FUNCTION_BLOCK "sq_carousel_st1"   // FB39, GRAPH
VERSION : 0.1
// stored: AcknowledgeErrorsRequired true, AutoNumber true, GraphVersion 6.0, InitialValuesAcquisition false, IsIECCheckEnabled false, LanguageInNetworks LAD, LockOperatingMode false, PermanentILProcessingInMANMode false, SetENOAutomatically false, SkipSteps false, UDAEnableTagReadback false, WithAlarmHandling true
   // inherited from GRAPH_BASE
   VAR
      OFF_SQ_BASE : Bool;
   END_VAR
   VAR_INPUT
      OFF_SQ { ExternalAccessible := 'False'; ExternalVisible := 'False'; ExternalWritable := 'False'} : Bool := false;   // Turn sequence off
      INIT_SQ { ExternalAccessible := 'False'; ExternalVisible := 'False'; ExternalWritable := 'False'} : Bool := false;   // Set sequence to initial state
      ACK_EF { ExternalAccessible := 'False'; ExternalVisible := 'False'; ExternalWritable := 'False'} : Bool := false;   // Acknowledge all errors and faults
      S_PREV { ExternalAccessible := 'False'; ExternalVisible := 'False'; ExternalWritable := 'False'} : Bool := false;   // Output previous step in parameter S_NO
      S_NEXT { ExternalAccessible := 'False'; ExternalVisible := 'False'; ExternalWritable := 'False'} : Bool := false;   // Indicate next step in parameter S_NO
      SW_AUTO { ExternalAccessible := 'False'; ExternalVisible := 'False'; ExternalWritable := 'False'} : Bool := false;   // Automatic mode
      SW_TAP { ExternalAccessible := 'False'; ExternalVisible := 'False'; ExternalWritable := 'False'} : Bool := false;   // Semiautomatic/switch with transition
      SW_TOP { ExternalAccessible := 'False'; ExternalVisible := 'False'; ExternalWritable := 'False'} : Bool := false;   // Semiautomatic/ignore transition
      SW_MAN { ExternalAccessible := 'False'; ExternalVisible := 'False'; ExternalWritable := 'False'} : Bool := false;   // Manual mode
      S_SEL { ExternalAccessible := 'False'; ExternalVisible := 'False'; ExternalWritable := 'False'} : Int := 0;   // Select step to be output to S_NO
      S_ON { ExternalAccessible := 'False'; ExternalVisible := 'False'; ExternalWritable := 'False'} : Bool := false;   // Activate step indicated in S_NO
      S_OFF { ExternalAccessible := 'False'; ExternalVisible := 'False'; ExternalWritable := 'False'} : Bool := false;   // Deactivate step indicated S_NO
      T_PUSH { ExternalAccessible := 'False'; ExternalVisible := 'False'; ExternalWritable := 'False'} : Bool := false;   // Enable transition to switch in semi automatic mode
   END_VAR
   VAR_OUTPUT
      S_NO { ExternalAccessible := 'False'; ExternalVisible := 'False'; ExternalWritable := 'False'} : Int := 0;   // Step number
      S_MORE { ExternalAccessible := 'False'; ExternalVisible := 'False'; ExternalWritable := 'False'} : Bool := false;   // More steps are available and can be shown in S_NO
      S_ACTIVE { ExternalAccessible := 'False'; ExternalVisible := 'False'; ExternalWritable := 'False'} : Bool := false;   // Step indicated in S_NO is active
      ERR_FLT { ExternalAccessible := 'False'; ExternalVisible := 'False'; ExternalWritable := 'False'} : Bool := false;   // Interlock or supervision group error
      AUTO_ON { ExternalAccessible := 'False'; ExternalVisible := 'False'; ExternalWritable := 'False'} : Bool := false;   // Automatic mode is active
      TAP_ON { ExternalAccessible := 'False'; ExternalVisible := 'False'; ExternalWritable := 'False'} : Bool := false;   // Semiautomatic mode/step with transition enabled
      TOP_ON { ExternalAccessible := 'False'; ExternalVisible := 'False'; ExternalWritable := 'False'} : Bool := false;   // Semiautomatic mode/ignore transition enabled
      MAN_ON { ExternalAccessible := 'False'; ExternalVisible := 'False'; ExternalWritable := 'False'} : Bool := false;   // Manual mode is active
   END_VAR
   VAR
      dummy : Bool;
      start : Bool;
      base : Bool;
      startEmpty : Bool;
   END_VAR
   VAR_TEMP   // added for the SCL form of the ladder/FBD networks
      _w1 : Bool;
      _w2 : Bool;
   END_VAR
BEGIN
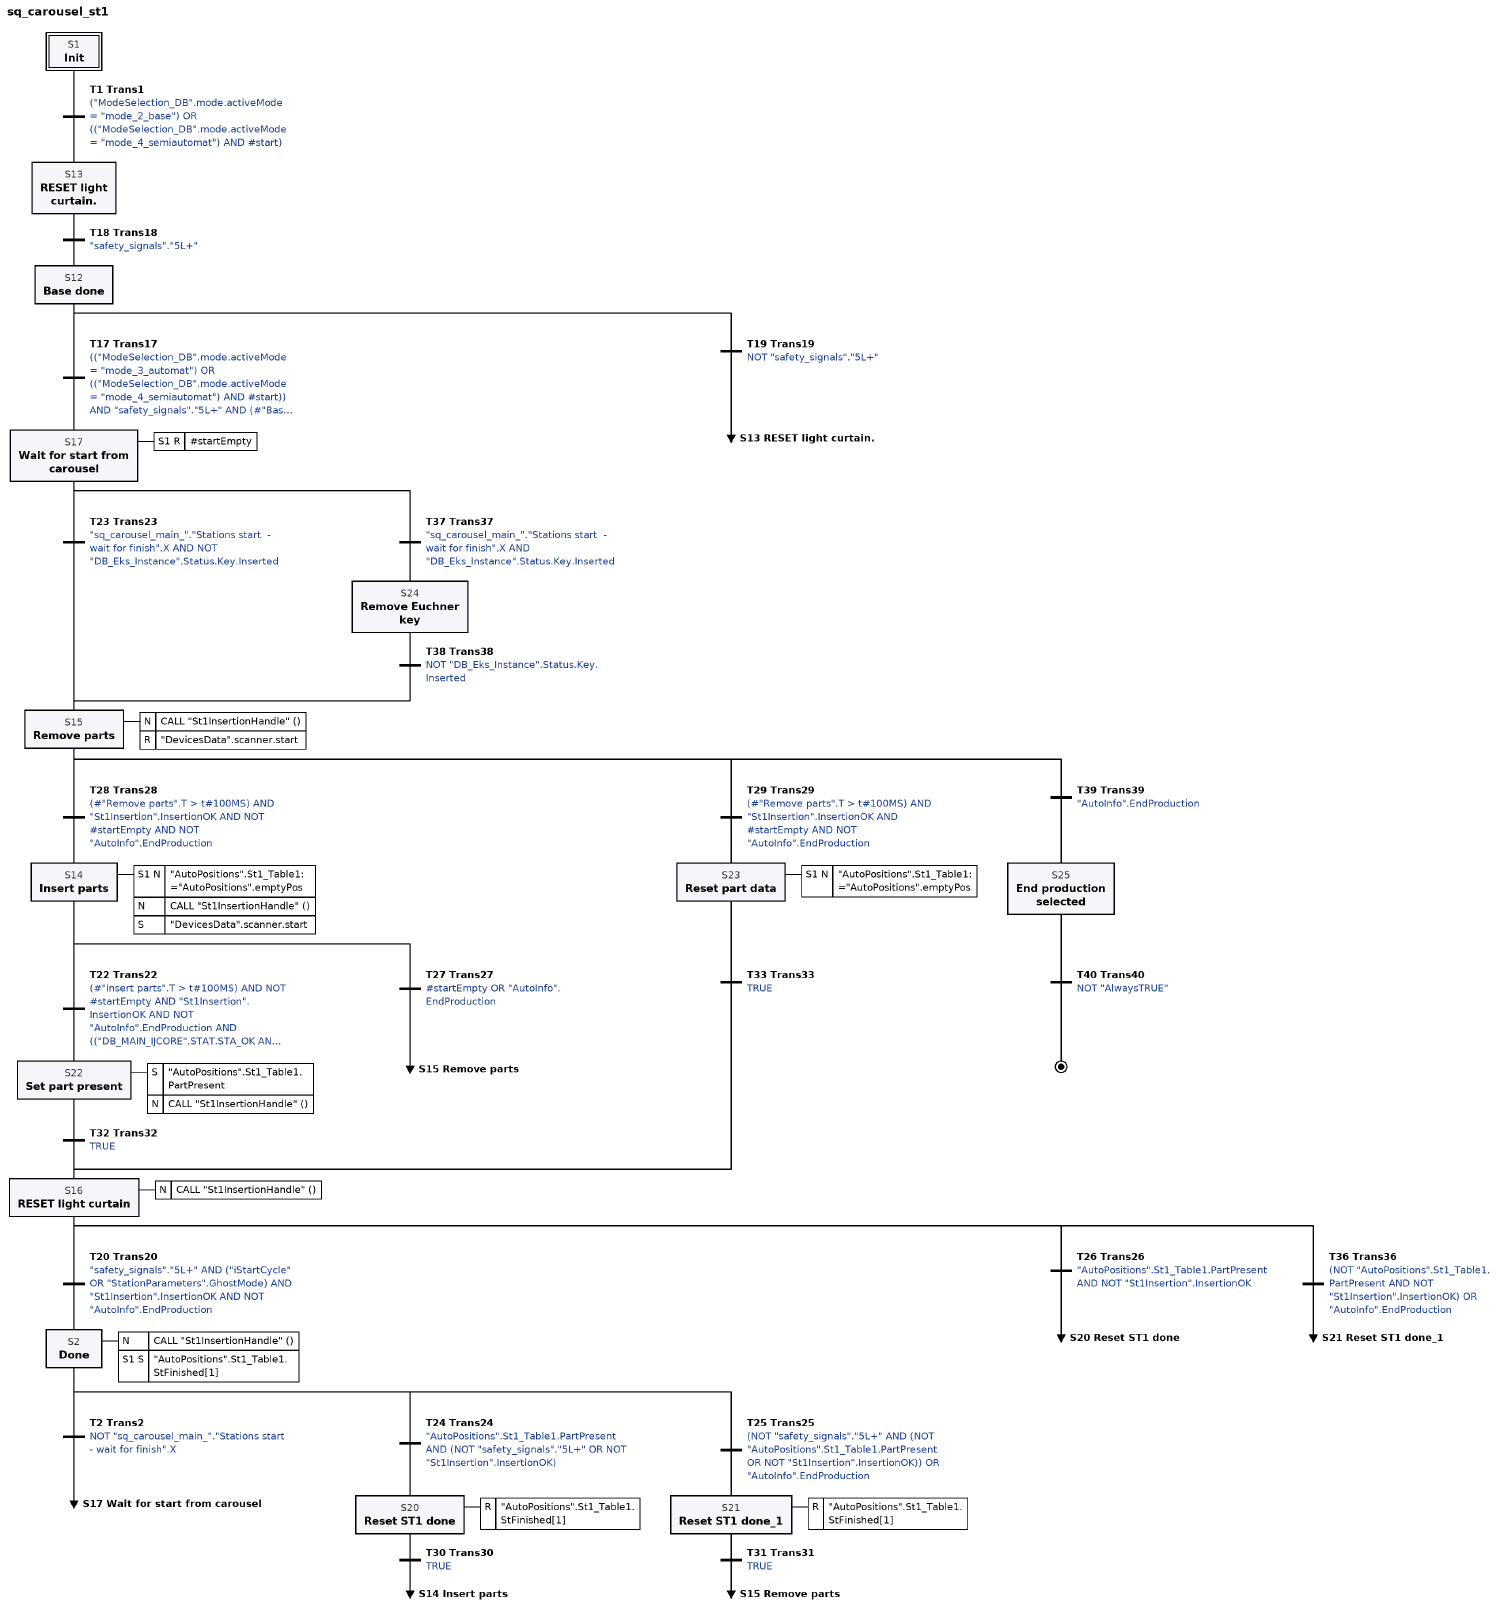
   // permanent pre-instructions
   NETWORK 1
      #base := TRUE;
   NETWORK 2
      "St1Insertion".ExpectedSensors := "St1Insertion".EmptyBits;
      #_w1 := ("ModeSelection_DB".mode.activeMode = "mode_3_automat") OR ("ModeSelection_DB".mode.activeMode = "mode_4_semiautomat");
      IF #_w1 THEN "St1Insertion".UsedSensors := "St1Insertion".FullBits; END_IF;
      IF NOT #_w1 THEN "St1Insertion".UsedSensors := "St1Insertion".EmptyBits; END_IF;
      #_w2 := ("AutoPositions".St1_Table1.PartPresent OR #"Insert parts".X) AND NOT #startEmpty AND NOT "StationParameters".GhostMode AND NOT #"Remove parts".X;
      IF #_w2 THEN
          MOVE_BLK(IN := "DB_ProductionProgramActual".Program.St1Insertion[1],
                   COUNT := 20,
                   OUT => "St1Insertion".ExpectedSensors[1]);
          MOVE_BLK(IN := "DB_ProductionProgramActual".Program.St1InsertionUsed[1],
                   COUNT := 20,
                   OUT => "St1Insertion".UsedSensors[1]);
      END_IF;
      "St1InsertionHandle"();

   // sequencer 1
   INITIAL_STEP Init:   // S1, max time T#10S, warning time T#7S
   END_STEP
   TRANSITION Trans1 FROM Init TO "RESET light curtain."   // T1
      := ("ModeSelection_DB".mode.activeMode = "mode_2_base") OR (("ModeSelection_DB".mode.activeMode = "mode_4_semiautomat") AND #start);
   END_TRANSITION
   STEP Done:   // S2, max time T#10S, warning time T#7S
              N    CALL "St1InsertionHandle" ()
          S1  S    "AutoPositions".St1_Table1.StFinished[1]
   END_STEP
   TRANSITION Trans2 FROM Done TO "Wait for start from carousel"   // T2, jump
      := NOT "sq_carousel_main_"."Stations start  - wait for finish".X;
   END_TRANSITION
   TRANSITION Trans24 FROM Done TO "Reset ST1 done"   // T24
      := "AutoPositions".St1_Table1.PartPresent AND (NOT "safety_signals"."5L+" OR NOT "St1Insertion".InsertionOK);
   END_TRANSITION
   TRANSITION Trans25 FROM Done TO "Reset ST1 done_1"   // T25
      := (NOT "safety_signals"."5L+" AND (NOT "AutoPositions".St1_Table1.PartPresent OR NOT "St1Insertion".InsertionOK)) OR "AutoInfo".EndProduction;
   END_TRANSITION
   STEP "Base done":   // S12, max time T#10S, warning time T#7S
   END_STEP
   TRANSITION Trans17 FROM "Base done" TO "Wait for start from carousel"   // T17
      := (("ModeSelection_DB".mode.activeMode = "mode_3_automat") OR (("ModeSelection_DB".mode.activeMode = "mode_4_semiautomat") AND #start)) AND "safety_signals"."5L+" AND (#"Base done".T > t#2000MS);
   END_TRANSITION
   TRANSITION Trans19 FROM "Base done" TO "RESET light curtain."   // T19, jump
      := NOT "safety_signals"."5L+";
   END_TRANSITION
   STEP "RESET light curtain.":   // S13, max time T#10S, warning time T#7S
   END_STEP
   TRANSITION Trans18 FROM "RESET light curtain." TO "Base done"   // T18
      := "safety_signals"."5L+";
   END_TRANSITION
   STEP "Insert parts":   // S14, max time T#10S, warning time T#7S
          S1  N    "AutoPositions".St1_Table1:="AutoPositions".emptyPos
              N    CALL "St1InsertionHandle" ()
              S    "DevicesData".scanner.start
   END_STEP
   TRANSITION Trans22 FROM "Insert parts" TO "Set part present"   // T22
      := (#"Insert parts".T > t#100MS) AND NOT #startEmpty AND "St1Insertion".InsertionOK AND NOT "AutoInfo".EndProduction AND (("DB_MAIN_IJCORE".STAT.STA_OK AND "DB_MAIN_IJCORE".STAT.TRC_OK) OR NOT "DB_MAIN_IJCORE".Enable);
   END_TRANSITION
   TRANSITION Trans27 FROM "Insert parts" TO "Remove parts"   // T27, jump
      := #startEmpty OR "AutoInfo".EndProduction;
   END_TRANSITION
   STEP "Remove parts":   // S15, max time T#10S, warning time T#7S
              N    CALL "St1InsertionHandle" ()
              R    "DevicesData".scanner.start
   END_STEP
   TRANSITION Trans28 FROM "Remove parts" TO "Insert parts"   // T28
      := (#"Remove parts".T > t#100MS) AND "St1Insertion".InsertionOK AND NOT #startEmpty AND NOT "AutoInfo".EndProduction;
   END_TRANSITION
   TRANSITION Trans29 FROM "Remove parts" TO "Reset part data"   // T29
      := (#"Remove parts".T > t#100MS) AND "St1Insertion".InsertionOK AND #startEmpty AND NOT "AutoInfo".EndProduction;
   END_TRANSITION
   TRANSITION Trans39 FROM "Remove parts" TO "End production selected"   // T39
      := "AutoInfo".EndProduction;
   END_TRANSITION
   STEP "RESET light curtain":   // S16, max time T#10S, warning time T#7S
              N    CALL "St1InsertionHandle" ()
   END_STEP
   TRANSITION Trans20 FROM "RESET light curtain" TO Done   // T20
      := "safety_signals"."5L+" AND ("iStartCycle" OR "StationParameters".GhostMode) AND "St1Insertion".InsertionOK AND NOT "AutoInfo".EndProduction;
   END_TRANSITION
   TRANSITION Trans26 FROM "RESET light curtain" TO "Reset ST1 done"   // T26, jump
      := "AutoPositions".St1_Table1.PartPresent AND NOT "St1Insertion".InsertionOK;
   END_TRANSITION
   TRANSITION Trans36 FROM "RESET light curtain" TO "Reset ST1 done_1"   // T36, jump
      := (NOT "AutoPositions".St1_Table1.PartPresent AND NOT "St1Insertion".InsertionOK) OR "AutoInfo".EndProduction;
   END_TRANSITION
   STEP "Wait for start from carousel":   // S17, max time T#10S, warning time T#7S
          S1  R    #startEmpty
   END_STEP
   TRANSITION Trans23 FROM "Wait for start from carousel" TO "Remove parts"   // T23
      := "sq_carousel_main_"."Stations start  - wait for finish".X AND NOT "DB_Eks_Instance".Status.Key.Inserted;
   END_TRANSITION
   TRANSITION Trans37 FROM "Wait for start from carousel" TO "Remove Euchner key"   // T37
      := "sq_carousel_main_"."Stations start  - wait for finish".X AND "DB_Eks_Instance".Status.Key.Inserted;
   END_TRANSITION
   STEP "Reset ST1 done":   // S20, max time T#10S, warning time T#7S
              R    "AutoPositions".St1_Table1.StFinished[1]
   END_STEP
   TRANSITION Trans30 FROM "Reset ST1 done" TO "Insert parts"   // T30, jump
      := TRUE;
   END_TRANSITION
   STEP "Reset ST1 done_1":   // S21, max time T#10S, warning time T#7S
              R    "AutoPositions".St1_Table1.StFinished[1]
   END_STEP
   TRANSITION Trans31 FROM "Reset ST1 done_1" TO "Remove parts"   // T31, jump
      := TRUE;
   END_TRANSITION
   STEP "Set part present":   // S22, max time T#10S, warning time T#7S
              S    "AutoPositions".St1_Table1.PartPresent
              N    CALL "St1InsertionHandle" ()
   END_STEP
   TRANSITION Trans32 FROM "Set part present" TO "RESET light curtain"   // T32
      := TRUE;
   END_TRANSITION
   STEP "Reset part data":   // S23, max time T#10S, warning time T#7S
          S1  N    "AutoPositions".St1_Table1:="AutoPositions".emptyPos
   END_STEP
   TRANSITION Trans33 FROM "Reset part data" TO "RESET light curtain"   // T33
      := TRUE;
   END_TRANSITION
   STEP "Remove Euchner key":   // S24, max time T#10S, warning time T#7S
   END_STEP
   TRANSITION Trans38 FROM "Remove Euchner key" TO "Remove parts"   // T38
      := NOT "DB_Eks_Instance".Status.Key.Inserted;
   END_TRANSITION
   STEP "End production selected":   // S25, max time T#10S, warning time T#7S
   END_STEP
   TRANSITION Trans40 FROM "End production selected" TO END   // T40
      := NOT "AlwaysTRUE";
   END_TRANSITION
END_FUNCTION_BLOCK

FUNCTION "St1InsertionHandle" : Void
{ S7_Optimized_Access := 'TRUE' }
VERSION : 0.1
   VAR_TEMP 
      i : Int;
      res : Bool;
      empty : Bool;
      lastNOKIndex : Int;
   END_VAR


BEGIN
	
	#i := 1;
	"St1Insertion".SensorsState[#i] := "DevicesData".Camera[1].Result = 1;
	#i := #i + 1;
	"St1Insertion".SensorsState[#i] := "DevicesData".Camera[2].Result = 1;
	#i := #i + 1;
	"St1Insertion".SensorsState[#i] := "DevicesData".Camera[3].Result = 1;
	#i := #i + 1;
	"St1Insertion".SensorsState[#i] := "DevicesData".Camera[4].Result = 1;
	#i := #i + 1;
	"St1Insertion".SensorsState[#i] := "DB_INST_READINGS".Reading[1].OK = 1;
	#i := #i + 1;
	"St1Insertion".SensorsState[#i] := "DB_INST_READINGS".Reading[2].OK = 1;
	#i := #i + 1;
	"St1Insertion".SensorsState[#i] := "DB_INST_READINGS".Reading[3].OK = 1;
	#i := #i + 1;
	"St1Insertion".SensorsState[#i] := "DB_INST_READINGS".Reading[4].OK = 1;
	#i := #i + 1;
	"St1Insertion".SensorsState[#i] := "DB_INST_READINGS".Reading[5].OK = 1;
	#i := #i + 1;
	"St1Insertion".SensorsState[#i] := "DB_INST_READINGS".Reading[6].OK = 1;
	#i := #i + 1;
	"St1Insertion".SensorsState[#i] := "DB_INST_READINGS".Reading[7].OK = 1;
	#i := #i + 1;
	"St1Insertion".SensorsState[#i] := "DB_INST_READINGS".Reading[8].OK = 1;
	#i := #i + 1;
	"St1Insertion".SensorsState[#i] := FALSE;
	#i := #i + 1;
	"St1Insertion".SensorsState[#i] := FALSE;
	#i := #i + 1;
	"St1Insertion".SensorsState[#i] := FALSE;
	#i := #i + 1;
	"St1Insertion".SensorsState[#i] := FALSE;
	#i := #i + 1;
	"St1Insertion".SensorsState[#i] := FALSE;
	#i := #i + 1;
	"St1Insertion".SensorsState[#i] := "Sensor_LH_PP" = 1;
	#i := #i + 1;
	"St1Insertion".SensorsState[#i] := "Sensor_RH_PP" = 1;
	
	#lastNOKIndex := 1;
	
	#res := TRUE;
	#empty := true;
	FOR #i := 1 TO 20 DO
	    
	    //Check if all sensors are zero
	    IF "St1Insertion".SensorsState[#i] THEN
	        #empty := false;
	    END_IF;
	    //Check if sensor is correct
	    IF ("St1Insertion".SensorsState[#i] <> "St1Insertion".ExpectedSensors[#i]) AND
	            "St1Insertion".UsedSensors[#i] THEN
	            #res := false;
	            "St1Insertion".SensorsNOK[#i] := true;
	            "St1Insertion".NOKList[#lastNOKIndex] := #i;
	            #lastNOKIndex := #lastNOKIndex + 1;
	        ELSE
	            "St1Insertion".SensorsNOK[#i] := false;
	    END_IF;
	END_FOR;
	    
	//Reset rest of nok list
	FOR #i := #lastNOKIndex TO 20 DO
	        "St1Insertion".NOKList[#i] := 0;
	END_FOR;
	
	"St1Insertion".InsertionOK := #res;
	"St1Insertion".InsertionNOK := NOT #empty AND NOT #res;
	"St1Insertion".InsertionEmpty := #empty;
	
	
	
END_FUNCTION

FUNCTION_BLOCK "sq_carousel_st2"   // FB43, GRAPH
VERSION : 0.1
// stored: AcknowledgeErrorsRequired true, AutoNumber true, GraphVersion 6.0, InitialValuesAcquisition false, IsIECCheckEnabled false, LanguageInNetworks LAD, LockOperatingMode false, PermanentILProcessingInMANMode false, SetENOAutomatically false, SkipSteps false, UDAEnableTagReadback false, WithAlarmHandling true
   // inherited from GRAPH_BASE
   VAR
      OFF_SQ_BASE : Bool;
   END_VAR
   VAR_INPUT
      OFF_SQ { ExternalAccessible := 'False'; ExternalVisible := 'False'; ExternalWritable := 'False'} : Bool := false;   // Turn sequence off
      INIT_SQ { ExternalAccessible := 'False'; ExternalVisible := 'False'; ExternalWritable := 'False'} : Bool := false;   // Set sequence to initial state
      ACK_EF { ExternalAccessible := 'False'; ExternalVisible := 'False'; ExternalWritable := 'False'} : Bool := false;   // Acknowledge all errors and faults
      S_PREV { ExternalAccessible := 'False'; ExternalVisible := 'False'; ExternalWritable := 'False'} : Bool := false;   // Output previous step in parameter S_NO
      S_NEXT { ExternalAccessible := 'False'; ExternalVisible := 'False'; ExternalWritable := 'False'} : Bool := false;   // Indicate next step in parameter S_NO
      SW_AUTO { ExternalAccessible := 'False'; ExternalVisible := 'False'; ExternalWritable := 'False'} : Bool := false;   // Automatic mode
      SW_TAP { ExternalAccessible := 'False'; ExternalVisible := 'False'; ExternalWritable := 'False'} : Bool := false;   // Semiautomatic/switch with transition
      SW_TOP { ExternalAccessible := 'False'; ExternalVisible := 'False'; ExternalWritable := 'False'} : Bool := false;   // Semiautomatic/ignore transition
      SW_MAN { ExternalAccessible := 'False'; ExternalVisible := 'False'; ExternalWritable := 'False'} : Bool := false;   // Manual mode
      S_SEL { ExternalAccessible := 'False'; ExternalVisible := 'False'; ExternalWritable := 'False'} : Int := 0;   // Select step to be output to S_NO
      S_ON { ExternalAccessible := 'False'; ExternalVisible := 'False'; ExternalWritable := 'False'} : Bool := false;   // Activate step indicated in S_NO
      S_OFF { ExternalAccessible := 'False'; ExternalVisible := 'False'; ExternalWritable := 'False'} : Bool := false;   // Deactivate step indicated S_NO
      T_PUSH { ExternalAccessible := 'False'; ExternalVisible := 'False'; ExternalWritable := 'False'} : Bool := false;   // Enable transition to switch in semi automatic mode
   END_VAR
   VAR_OUTPUT
      S_NO { ExternalAccessible := 'False'; ExternalVisible := 'False'; ExternalWritable := 'False'} : Int := 0;   // Step number
      S_MORE { ExternalAccessible := 'False'; ExternalVisible := 'False'; ExternalWritable := 'False'} : Bool := false;   // More steps are available and can be shown in S_NO
      S_ACTIVE { ExternalAccessible := 'False'; ExternalVisible := 'False'; ExternalWritable := 'False'} : Bool := false;   // Step indicated in S_NO is active
      ERR_FLT { ExternalAccessible := 'False'; ExternalVisible := 'False'; ExternalWritable := 'False'} : Bool := false;   // Interlock or supervision group error
      AUTO_ON { ExternalAccessible := 'False'; ExternalVisible := 'False'; ExternalWritable := 'False'} : Bool := false;   // Automatic mode is active
      TAP_ON { ExternalAccessible := 'False'; ExternalVisible := 'False'; ExternalWritable := 'False'} : Bool := false;   // Semiautomatic mode/step with transition enabled
      TOP_ON { ExternalAccessible := 'False'; ExternalVisible := 'False'; ExternalWritable := 'False'} : Bool := false;   // Semiautomatic mode/ignore transition enabled
      MAN_ON { ExternalAccessible := 'False'; ExternalVisible := 'False'; ExternalWritable := 'False'} : Bool := false;   // Manual mode is active
   END_VAR
   VAR
      dummy : Bool;
      start : Bool;
      base : Bool;
   END_VAR
BEGIN
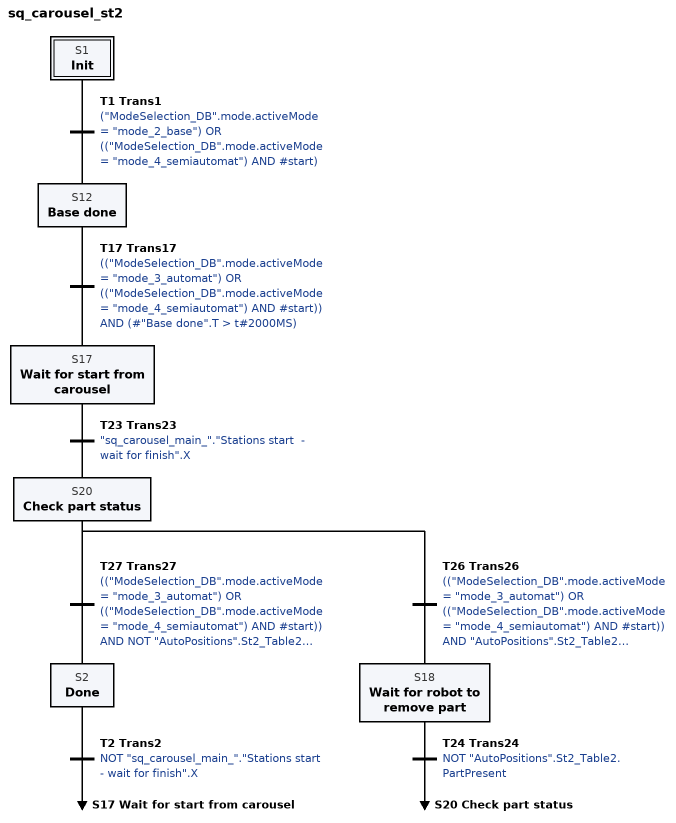
   // permanent pre-instructions
   NETWORK 1
   TITLE = base position
      #base := TRUE;

   // sequencer 1
   INITIAL_STEP Init:   // S1, max time T#10S, warning time T#7S
   END_STEP
   TRANSITION Trans1 FROM Init TO "Base done"   // T1
      := ("ModeSelection_DB".mode.activeMode = "mode_2_base") OR (("ModeSelection_DB".mode.activeMode = "mode_4_semiautomat") AND #start);
   END_TRANSITION
   STEP Done:   // S2, max time T#10S, warning time T#7S
   END_STEP
   TRANSITION Trans2 FROM Done TO "Wait for start from carousel"   // T2, jump
      := NOT "sq_carousel_main_"."Stations start  - wait for finish".X;
   END_TRANSITION
   STEP "Base done":   // S12, max time T#10S, warning time T#7S
   END_STEP
   TRANSITION Trans17 FROM "Base done" TO "Wait for start from carousel"   // T17
      := (("ModeSelection_DB".mode.activeMode = "mode_3_automat") OR (("ModeSelection_DB".mode.activeMode = "mode_4_semiautomat") AND #start)) AND (#"Base done".T > t#2000MS);
   END_TRANSITION
   STEP "Wait for start from carousel":   // S17, max time T#10S, warning time T#7S
   END_STEP
   TRANSITION Trans23 FROM "Wait for start from carousel" TO "Check part status"   // T23
      := "sq_carousel_main_"."Stations start  - wait for finish".X;
   END_TRANSITION
   STEP "Check part status":   // S20, max time T#10S, warning time T#7S
   END_STEP
   TRANSITION Trans27 FROM "Check part status" TO Done   // T27
      := (("ModeSelection_DB".mode.activeMode = "mode_3_automat") OR (("ModeSelection_DB".mode.activeMode = "mode_4_semiautomat") AND #start)) AND NOT "AutoPositions".St2_Table2.PartPresent AND "iR1OutOfSt2";
   END_TRANSITION
   TRANSITION Trans26 FROM "Check part status" TO "Wait for robot to remove part"   // T26
      := (("ModeSelection_DB".mode.activeMode = "mode_3_automat") OR (("ModeSelection_DB".mode.activeMode = "mode_4_semiautomat") AND #start)) AND "AutoPositions".St2_Table2.PartPresent;
   END_TRANSITION
   STEP "Wait for robot to remove part":   // S18, max time T#10S, warning time T#7S
   END_STEP
   TRANSITION Trans24 FROM "Wait for robot to remove part" TO "Check part status"   // T24, jump
      := NOT "AutoPositions".St2_Table2.PartPresent;
   END_TRANSITION
END_FUNCTION_BLOCK

FUNCTION_BLOCK "sq_jig"   // FB41, GRAPH
VERSION : 0.1
// stored: AcknowledgeErrorsRequired true, AutoNumber true, GraphVersion 6.0, InitialValuesAcquisition false, IsIECCheckEnabled false, LanguageInNetworks LAD, LockOperatingMode false, PermanentILProcessingInMANMode false, SetENOAutomatically false, SkipSteps false, UDAEnableTagReadback false, WithAlarmHandling true
   // inherited from GRAPH_BASE
   VAR
      OFF_SQ_BASE : Bool;
   END_VAR
   VAR_INPUT
      OFF_SQ { ExternalAccessible := 'False'; ExternalVisible := 'False'; ExternalWritable := 'False'} : Bool := false;   // Turn sequence off
      INIT_SQ { ExternalAccessible := 'False'; ExternalVisible := 'False'; ExternalWritable := 'False'} : Bool := false;   // Set sequence to initial state
      ACK_EF { ExternalAccessible := 'False'; ExternalVisible := 'False'; ExternalWritable := 'False'} : Bool := false;   // Acknowledge all errors and faults
      S_PREV { ExternalAccessible := 'False'; ExternalVisible := 'False'; ExternalWritable := 'False'} : Bool := false;   // Output previous step in parameter S_NO
      S_NEXT { ExternalAccessible := 'False'; ExternalVisible := 'False'; ExternalWritable := 'False'} : Bool := false;   // Indicate next step in parameter S_NO
      SW_AUTO { ExternalAccessible := 'False'; ExternalVisible := 'False'; ExternalWritable := 'False'} : Bool := false;   // Automatic mode
      SW_TAP { ExternalAccessible := 'False'; ExternalVisible := 'False'; ExternalWritable := 'False'} : Bool := false;   // Semiautomatic/switch with transition
      SW_TOP { ExternalAccessible := 'False'; ExternalVisible := 'False'; ExternalWritable := 'False'} : Bool := false;   // Semiautomatic/ignore transition
      SW_MAN { ExternalAccessible := 'False'; ExternalVisible := 'False'; ExternalWritable := 'False'} : Bool := false;   // Manual mode
      S_SEL { ExternalAccessible := 'False'; ExternalVisible := 'False'; ExternalWritable := 'False'} : Int := 0;   // Select step to be output to S_NO
      S_ON { ExternalAccessible := 'False'; ExternalVisible := 'False'; ExternalWritable := 'False'} : Bool := false;   // Activate step indicated in S_NO
      S_OFF { ExternalAccessible := 'False'; ExternalVisible := 'False'; ExternalWritable := 'False'} : Bool := false;   // Deactivate step indicated S_NO
      T_PUSH { ExternalAccessible := 'False'; ExternalVisible := 'False'; ExternalWritable := 'False'} : Bool := false;   // Enable transition to switch in semi automatic mode
   END_VAR
   VAR_OUTPUT
      S_NO { ExternalAccessible := 'False'; ExternalVisible := 'False'; ExternalWritable := 'False'} : Int := 0;   // Step number
      S_MORE { ExternalAccessible := 'False'; ExternalVisible := 'False'; ExternalWritable := 'False'} : Bool := false;   // More steps are available and can be shown in S_NO
      S_ACTIVE { ExternalAccessible := 'False'; ExternalVisible := 'False'; ExternalWritable := 'False'} : Bool := false;   // Step indicated in S_NO is active
      ERR_FLT { ExternalAccessible := 'False'; ExternalVisible := 'False'; ExternalWritable := 'False'} : Bool := false;   // Interlock or supervision group error
      AUTO_ON { ExternalAccessible := 'False'; ExternalVisible := 'False'; ExternalWritable := 'False'} : Bool := false;   // Automatic mode is active
      TAP_ON { ExternalAccessible := 'False'; ExternalVisible := 'False'; ExternalWritable := 'False'} : Bool := false;   // Semiautomatic mode/step with transition enabled
      TOP_ON { ExternalAccessible := 'False'; ExternalVisible := 'False'; ExternalWritable := 'False'} : Bool := false;   // Semiautomatic mode/ignore transition enabled
      MAN_ON { ExternalAccessible := 'False'; ExternalVisible := 'False'; ExternalWritable := 'False'} : Bool := false;   // Manual mode is active
   END_VAR
   VAR
      dummy : Bool;
      start : Bool;
      base : Bool;
   END_VAR
   VAR_TEMP   // added for the SCL form of the ladder/FBD networks
      _w1 : Bool;
   END_VAR
BEGIN
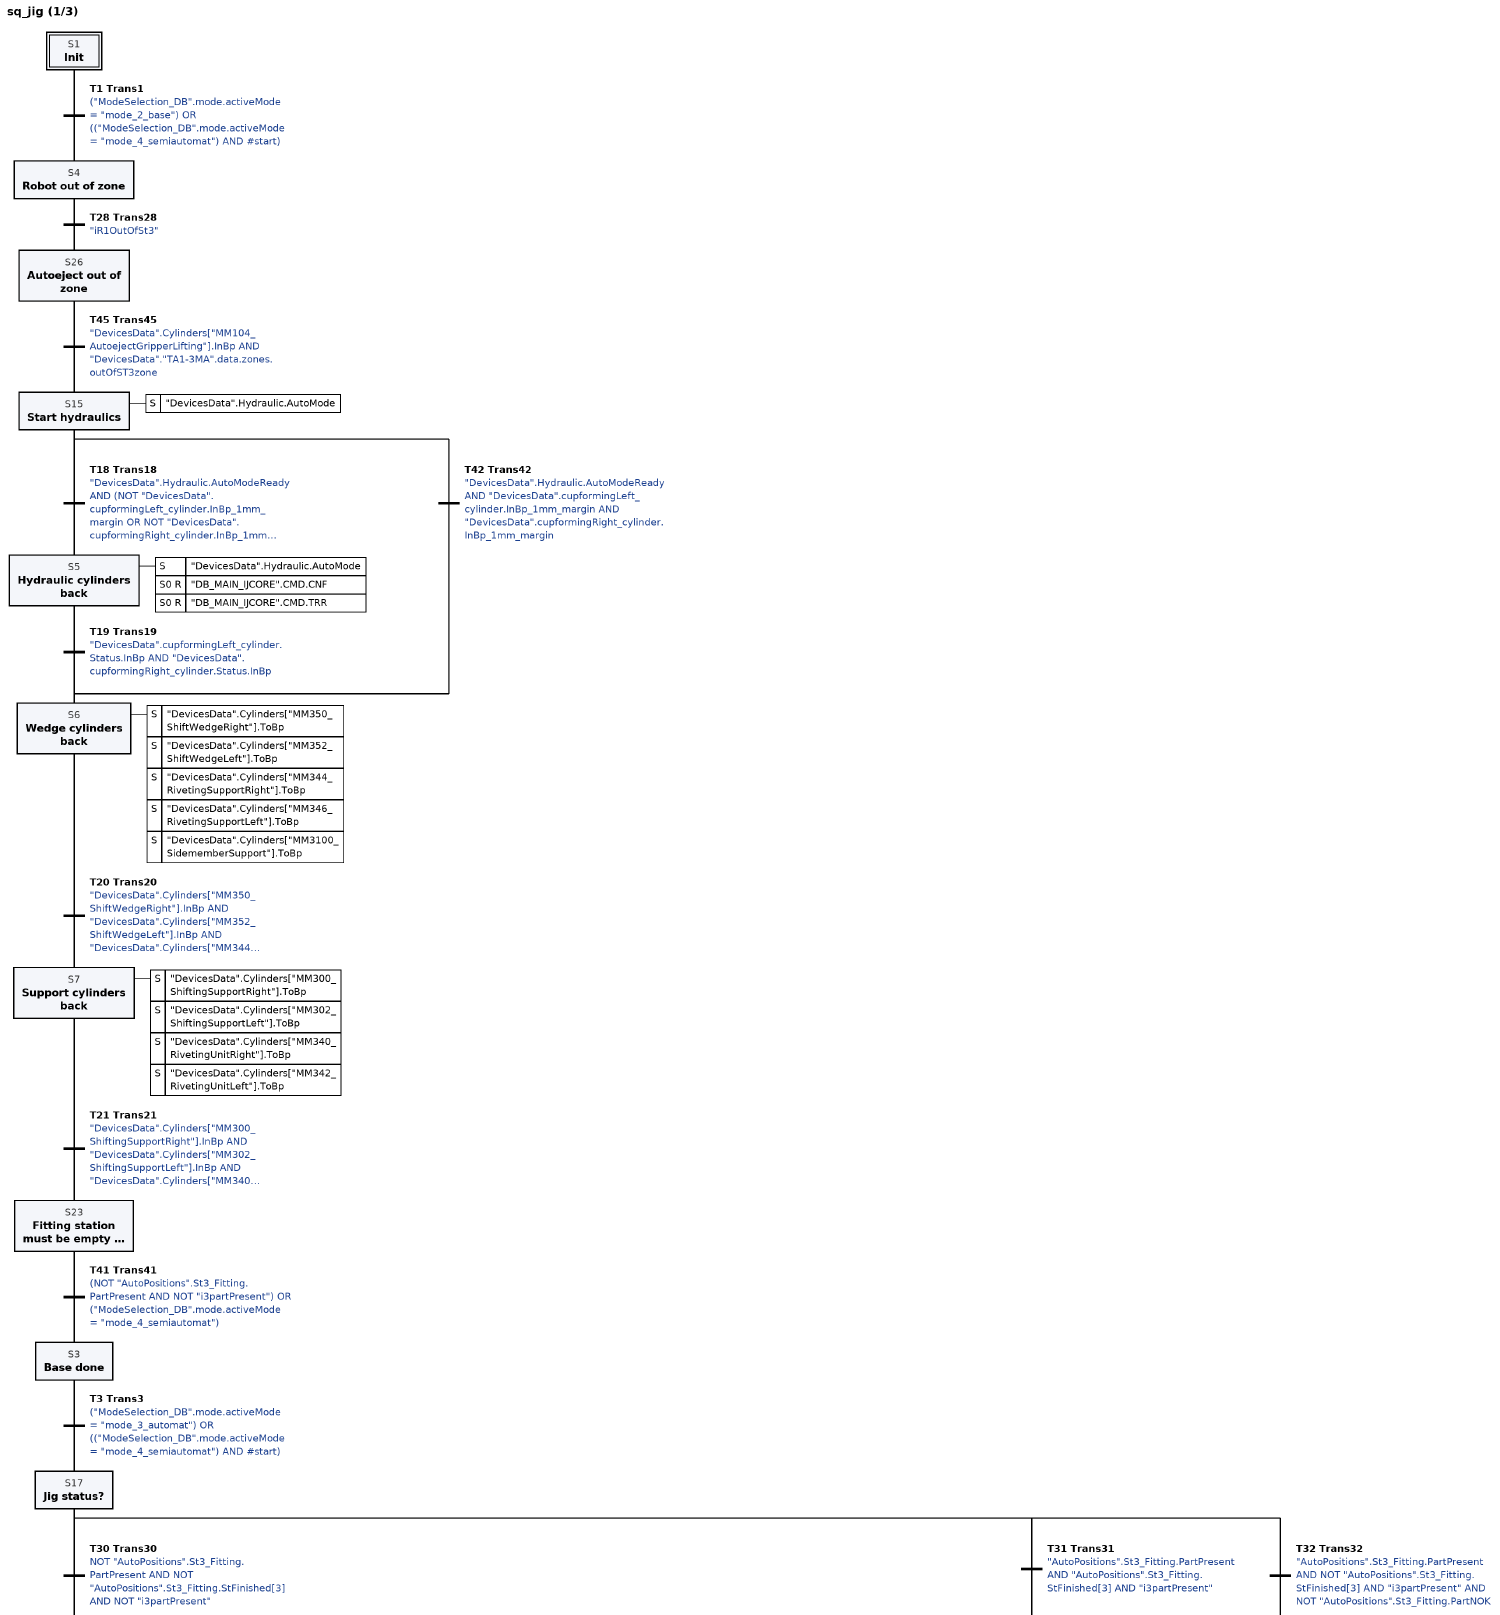
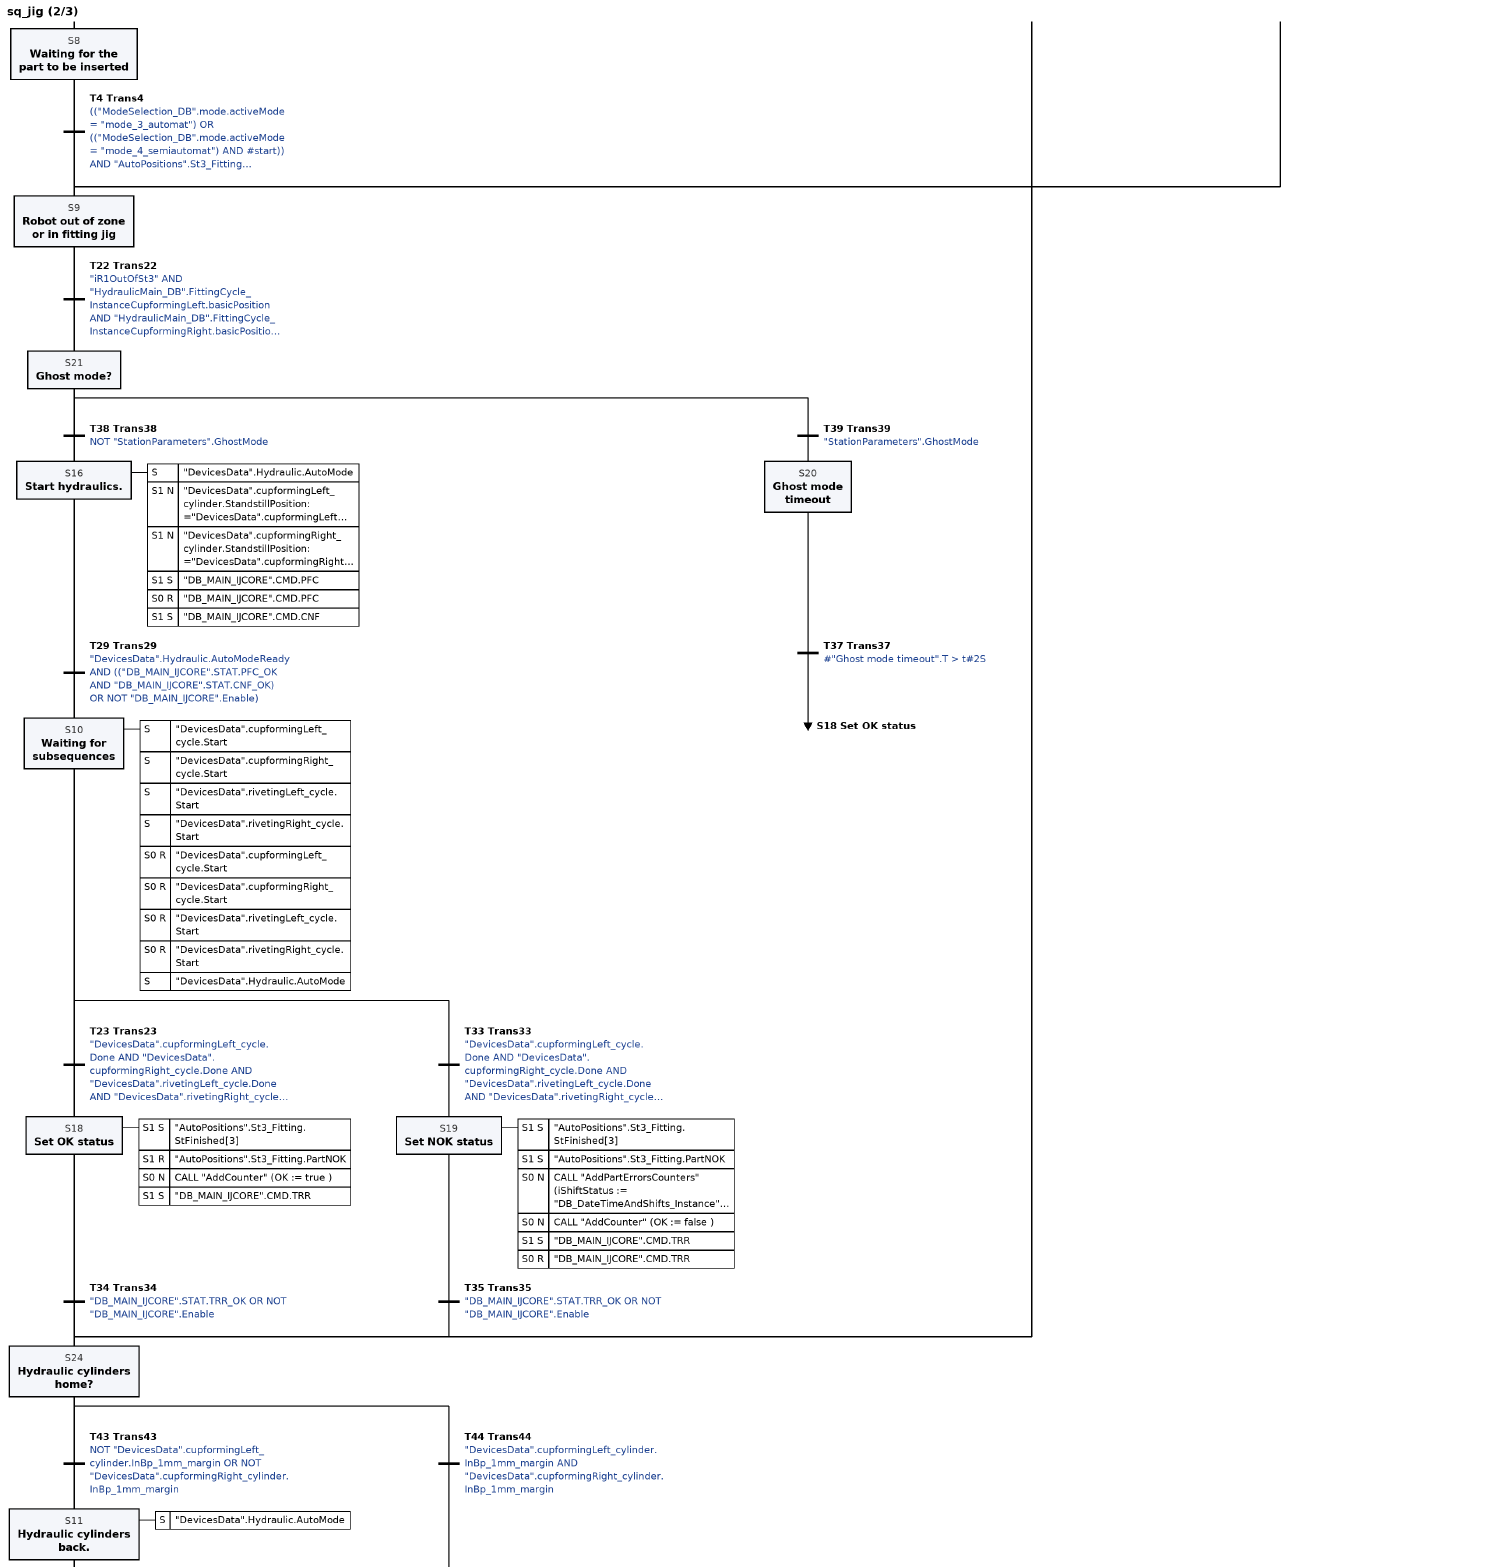
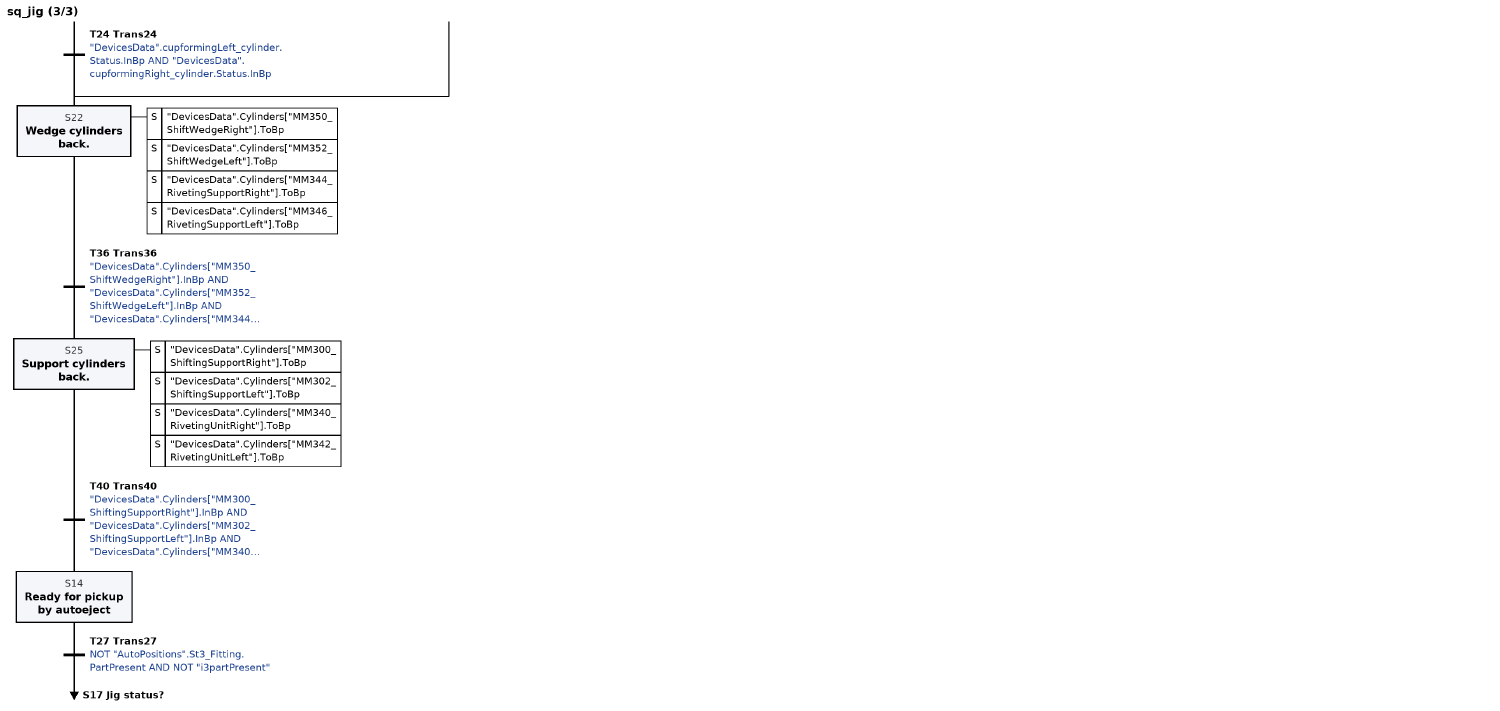
   // permanent pre-instructions
   NETWORK 1
   TITLE = base position
      #base := "HydraulicMain_DB".FittingCycle_InstanceCupformingLeft.basicPosition AND "HydraulicMain_DB".FittingCycle_InstanceCupformingRight.basicPosition AND "DB_Devices_Instance".RivetingCycleLeft_Instance.basicPosition AND "DB_Devices_Instance".RivetingCycleRight_Instance.basicPosition AND "DevicesData".Digiforce1.Ready AND "DevicesData".Digiforce1.programOK AND "DevicesData".Digiforce2.Ready AND "DevicesData".Digiforce2.programOK AND NOT "Devices_Diagnostic_DB".PNmissing;

   // sequencer 1
   INITIAL_STEP Init:   // S1, max time T#10S, warning time T#7S
   END_STEP
   TRANSITION Trans1 FROM Init TO "Robot out of zone"   // T1
      := ("ModeSelection_DB".mode.activeMode = "mode_2_base") OR (("ModeSelection_DB".mode.activeMode = "mode_4_semiautomat") AND #start);
   END_TRANSITION
   STEP "Start hydraulics":   // S15, max time T#10S, warning time T#7S
      supervision V := #"Start hydraulics".T > #"Start hydraulics".T_MAX;
              S    "DevicesData".Hydraulic.AutoMode
   END_STEP
   TRANSITION Trans18 FROM "Start hydraulics" TO "Hydraulic cylinders back"   // T18
      := "DevicesData".Hydraulic.AutoModeReady AND (NOT "DevicesData".cupformingLeft_cylinder.InBp_1mm_margin OR NOT "DevicesData".cupformingRight_cylinder.InBp_1mm_margin);
   END_TRANSITION
   TRANSITION Trans42 FROM "Start hydraulics" TO "Wedge cylinders back"   // T42
      := "DevicesData".Hydraulic.AutoModeReady AND "DevicesData".cupformingLeft_cylinder.InBp_1mm_margin AND "DevicesData".cupformingRight_cylinder.InBp_1mm_margin;
   END_TRANSITION
   STEP "Waiting for the part to be inserted":   // S8, max time T#10S, warning time T#7S
   END_STEP
   TRANSITION Trans4 FROM "Waiting for the part to be inserted" TO "Robot out of zone or in fitting jig"   // T4
      := (("ModeSelection_DB".mode.activeMode = "mode_3_automat") OR (("ModeSelection_DB".mode.activeMode = "mode_4_semiautomat") AND #start)) AND "AutoPositions".St3_Fitting.PartPresent AND NOT "AutoPositions".St3_Fitting.StFinished[3] AND ("i3partPresent" OR "StationParameters".GhostMode);
   END_TRANSITION
   STEP "Robot out of zone":   // S4, max time T#10S, warning time T#7S
      supervision V := #"Robot out of zone".T > #"Robot out of zone".T_MAX;
   END_STEP
   TRANSITION Trans28 FROM "Robot out of zone" TO "Autoeject out of zone"   // T28
      := "iR1OutOfSt3";
   END_TRANSITION
   STEP "Hydraulic cylinders back":   // S5, max time T#10S, warning time T#7S
      supervision V := #"Hydraulic cylinders back".T > #"Hydraulic cylinders back".T_MAX;
              S    "DevicesData".Hydraulic.AutoMode
          S0  R    "DB_MAIN_IJCORE".CMD.CNF
          S0  R    "DB_MAIN_IJCORE".CMD.TRR
   END_STEP
   TRANSITION Trans19 FROM "Hydraulic cylinders back" TO "Wedge cylinders back"   // T19
      := "DevicesData".cupformingLeft_cylinder.Status.InBp AND "DevicesData".cupformingRight_cylinder.Status.InBp;
   END_TRANSITION
   STEP "Wedge cylinders back":   // S6, max time T#10S, warning time T#7S
      supervision V := #"Wedge cylinders back".T > #"Wedge cylinders back".T_MAX;
              S    "DevicesData".Cylinders["MM350_ShiftWedgeRight"].ToBp
              S    "DevicesData".Cylinders["MM352_ShiftWedgeLeft"].ToBp
              S    "DevicesData".Cylinders["MM344_RivetingSupportRight"].ToBp
              S    "DevicesData".Cylinders["MM346_RivetingSupportLeft"].ToBp
              S    "DevicesData".Cylinders["MM3100_SidememberSupport"].ToBp
   END_STEP
   TRANSITION Trans20 FROM "Wedge cylinders back" TO "Support cylinders back"   // T20
      := "DevicesData".Cylinders["MM350_ShiftWedgeRight"].InBp AND "DevicesData".Cylinders["MM352_ShiftWedgeLeft"].InBp AND "DevicesData".Cylinders["MM344_RivetingSupportRight"].InBp AND "DevicesData".Cylinders["MM346_RivetingSupportLeft"].InBp AND "DevicesData".Cylinders["MM3100_SidememberSupport"].InBp;
   END_TRANSITION
   STEP "Support cylinders back":   // S7, max time T#10S, warning time T#7S
      supervision V := #"Support cylinders back".T > #"Support cylinders back".T_MAX;
              S    "DevicesData".Cylinders["MM300_ShiftingSupportRight"].ToBp
              S    "DevicesData".Cylinders["MM302_ShiftingSupportLeft"].ToBp
              S    "DevicesData".Cylinders["MM340_RivetingUnitRight"].ToBp
              S    "DevicesData".Cylinders["MM342_RivetingUnitLeft"].ToBp
   END_STEP
   TRANSITION Trans21 FROM "Support cylinders back" TO "Fitting station must be empty - remove part and delete status"   // T21
      := "DevicesData".Cylinders["MM300_ShiftingSupportRight"].InBp AND "DevicesData".Cylinders["MM302_ShiftingSupportLeft"].InBp AND "DevicesData".Cylinders["MM340_RivetingUnitRight"].InBp AND "DevicesData".Cylinders["MM342_RivetingUnitLeft"].InBp;
   END_TRANSITION
   STEP "Base done":   // S3, max time T#10S, warning time T#7S
   END_STEP
   TRANSITION Trans3 FROM "Base done" TO "Jig status?"   // T3
      := ("ModeSelection_DB".mode.activeMode = "mode_3_automat") OR (("ModeSelection_DB".mode.activeMode = "mode_4_semiautomat") AND #start);
   END_TRANSITION
   STEP "Robot out of zone or in fitting jig":   // S9, max time T#10S, warning time T#7S
      supervision V := #"Robot out of zone or in fitting jig".T > #"Robot out of zone or in fitting jig".T_MAX;
   END_STEP
   TRANSITION Trans22 FROM "Robot out of zone or in fitting jig" TO "Ghost mode?"   // T22
      := "iR1OutOfSt3" AND "HydraulicMain_DB".FittingCycle_InstanceCupformingLeft.basicPosition AND "HydraulicMain_DB".FittingCycle_InstanceCupformingRight.basicPosition AND "DB_Devices_Instance".RivetingCycleLeft_Instance.basicPosition AND "DB_Devices_Instance".RivetingCycleRight_Instance.basicPosition;
   END_TRANSITION
   STEP "Waiting for subsequences":   // S10, max time T#10S, warning time T#7S
              S    "DevicesData".cupformingLeft_cycle.Start
              S    "DevicesData".cupformingRight_cycle.Start
              S    "DevicesData".rivetingLeft_cycle.Start
              S    "DevicesData".rivetingRight_cycle.Start
          S0  R    "DevicesData".cupformingLeft_cycle.Start
          S0  R    "DevicesData".cupformingRight_cycle.Start
          S0  R    "DevicesData".rivetingLeft_cycle.Start
          S0  R    "DevicesData".rivetingRight_cycle.Start
              S    "DevicesData".Hydraulic.AutoMode
   END_STEP
   TRANSITION Trans23 FROM "Waiting for subsequences" TO "Set OK status"   // T23
      := "DevicesData".cupformingLeft_cycle.Done AND "DevicesData".cupformingRight_cycle.Done AND "DevicesData".rivetingLeft_cycle.Done AND "DevicesData".rivetingRight_cycle.Done AND "DevicesData".cupformingLeft_cycle.OK AND "DevicesData".cupformingRight_cycle.OK AND "DevicesData".rivetingLeft_cycle.OK AND "DevicesData".rivetingRight_cycle.OK;
   END_TRANSITION
   TRANSITION Trans33 FROM "Waiting for subsequences" TO "Set NOK status"   // T33
      := "DevicesData".cupformingLeft_cycle.Done AND "DevicesData".cupformingRight_cycle.Done AND "DevicesData".rivetingLeft_cycle.Done AND "DevicesData".rivetingRight_cycle.Done;
   END_TRANSITION
   STEP "Hydraulic cylinders back.":   // S11, max time T#10S, warning time T#7S
      supervision V := #"Hydraulic cylinders back.".T > #"Hydraulic cylinders back.".T_MAX;
              S    "DevicesData".Hydraulic.AutoMode
   END_STEP
   TRANSITION Trans24 FROM "Hydraulic cylinders back." TO "Wedge cylinders back."   // T24
      := "DevicesData".cupformingLeft_cylinder.Status.InBp AND "DevicesData".cupformingRight_cylinder.Status.InBp;
   END_TRANSITION
   STEP "Autoeject out of zone":   // S26, max time T#10S, warning time T#7S
      supervision V := #"Autoeject out of zone".T > #"Autoeject out of zone".T_MAX;
   END_STEP
   TRANSITION Trans45 FROM "Autoeject out of zone" TO "Start hydraulics"   // T45
      := "DevicesData".Cylinders["MM104_AutoejectGripperLifting"].InBp AND "DevicesData"."TA1-3MA".data.zones.outOfST3zone;
   END_TRANSITION
   STEP "Ready for pickup by autoeject":   // S14, max time T#10S, warning time T#7S
   END_STEP
   TRANSITION Trans27 FROM "Ready for pickup by autoeject" TO "Jig status?"   // T27, jump
      := NOT "AutoPositions".St3_Fitting.PartPresent AND NOT "i3partPresent";
   END_TRANSITION
   STEP "Start hydraulics.":   // S16, max time T#10S, warning time T#7S
      supervision V := #"Start hydraulics.".T > #"Start hydraulics.".T_MAX;
              S    "DevicesData".Hydraulic.AutoMode
          S1  N    "DevicesData".cupformingLeft_cylinder.StandstillPosition:="DevicesData".cupformingLeft_cylinder.Position
          S1  N    "DevicesData".cupformingRight_cylinder.StandstillPosition:="DevicesData".cupformingRight_cylinder.Position
          S1  S    "DB_MAIN_IJCORE".CMD.PFC
          S0  R    "DB_MAIN_IJCORE".CMD.PFC
          S1  S    "DB_MAIN_IJCORE".CMD.CNF
   END_STEP
   TRANSITION Trans29 FROM "Start hydraulics." TO "Waiting for subsequences"   // T29
      := "DevicesData".Hydraulic.AutoModeReady AND (("DB_MAIN_IJCORE".STAT.PFC_OK AND "DB_MAIN_IJCORE".STAT.CNF_OK) OR NOT "DB_MAIN_IJCORE".Enable);
   END_TRANSITION
   STEP "Jig status?":   // S17, max time T#10S, warning time T#7S
   END_STEP
   TRANSITION Trans30 FROM "Jig status?" TO "Waiting for the part to be inserted"   // T30
      := NOT "AutoPositions".St3_Fitting.PartPresent AND NOT "AutoPositions".St3_Fitting.StFinished[3] AND NOT "i3partPresent";
   END_TRANSITION
   TRANSITION Trans31 FROM "Jig status?" TO "Hydraulic cylinders home?"   // T31
      := "AutoPositions".St3_Fitting.PartPresent AND "AutoPositions".St3_Fitting.StFinished[3] AND "i3partPresent";
   END_TRANSITION
   TRANSITION Trans32 FROM "Jig status?" TO "Robot out of zone or in fitting jig"   // T32
      := "AutoPositions".St3_Fitting.PartPresent AND NOT "AutoPositions".St3_Fitting.StFinished[3] AND "i3partPresent" AND NOT "AutoPositions".St3_Fitting.PartNOK;
   END_TRANSITION
   STEP "Set OK status":   // S18, max time T#10S, warning time T#7S
          S1  S    "AutoPositions".St3_Fitting.StFinished[3]
          S1  R    "AutoPositions".St3_Fitting.PartNOK
          S0  N    CALL "AddCounter"
                   (OK := true
                   )
          S1  S    "DB_MAIN_IJCORE".CMD.TRR
   END_STEP
   TRANSITION Trans34 FROM "Set OK status" TO "Hydraulic cylinders home?"   // T34
      := "DB_MAIN_IJCORE".STAT.TRR_OK OR NOT "DB_MAIN_IJCORE".Enable;
   END_TRANSITION
   STEP "Set NOK status":   // S19, max time T#10S, warning time T#7S
          S1  S    "AutoPositions".St3_Fitting.StFinished[3]
          S1  S    "AutoPositions".St3_Fitting.PartNOK
          S0  N    CALL "AddPartErrorsCounters" (iShiftStatus := "DB_DateTimeAndShifts_Instance".ShiftStatus
                   )
          S0  N    CALL "AddCounter"
                   (OK := false
                   )
          S1  S    "DB_MAIN_IJCORE".CMD.TRR
          S0  R    "DB_MAIN_IJCORE".CMD.TRR
   END_STEP
   TRANSITION Trans35 FROM "Set NOK status" TO "Hydraulic cylinders home?"   // T35
      := "DB_MAIN_IJCORE".STAT.TRR_OK OR NOT "DB_MAIN_IJCORE".Enable;
   END_TRANSITION
   STEP "Ghost mode?":   // S21, max time T#10S, warning time T#7S
   END_STEP
   TRANSITION Trans38 FROM "Ghost mode?" TO "Start hydraulics."   // T38
      := NOT "StationParameters".GhostMode;
   END_TRANSITION
   TRANSITION Trans39 FROM "Ghost mode?" TO "Ghost mode timeout"   // T39
      := "StationParameters".GhostMode;
   END_TRANSITION
   STEP "Ghost mode timeout":   // S20, max time T#10S, warning time T#7S
   END_STEP
   TRANSITION Trans37 FROM "Ghost mode timeout" TO "Set OK status"   // T37, jump
      := #"Ghost mode timeout".T > t#2S;
   END_TRANSITION
   STEP "Fitting station must be empty - remove part and delete status":   // S23, max time T#2S, warning time T#7S
      supervision V := #"Fitting station must be empty - remove part and delete status".T > #"Fitting station must be empty - remove part and delete status".T_MAX;
   END_STEP
   TRANSITION Trans41 FROM "Fitting station must be empty - remove part and delete status" TO "Base done"   // T41
      := (NOT "AutoPositions".St3_Fitting.PartPresent AND NOT "i3partPresent") OR ("ModeSelection_DB".mode.activeMode = "mode_4_semiautomat");
   END_TRANSITION
   STEP "Hydraulic cylinders home?":   // S24, max time T#10S, warning time T#7S
   END_STEP
   TRANSITION Trans43 FROM "Hydraulic cylinders home?" TO "Hydraulic cylinders back."   // T43
      := NOT "DevicesData".cupformingLeft_cylinder.InBp_1mm_margin OR NOT "DevicesData".cupformingRight_cylinder.InBp_1mm_margin;
   END_TRANSITION
   TRANSITION Trans44 FROM "Hydraulic cylinders home?" TO "Wedge cylinders back."   // T44
      := "DevicesData".cupformingLeft_cylinder.InBp_1mm_margin AND "DevicesData".cupformingRight_cylinder.InBp_1mm_margin;
   END_TRANSITION
   STEP "Wedge cylinders back.":   // S22, max time T#10S, warning time T#7S
      supervision V := #"Wedge cylinders back.".T > #"Wedge cylinders back.".T_MAX;
              S    "DevicesData".Cylinders["MM350_ShiftWedgeRight"].ToBp
              S    "DevicesData".Cylinders["MM352_ShiftWedgeLeft"].ToBp
              S    "DevicesData".Cylinders["MM344_RivetingSupportRight"].ToBp
              S    "DevicesData".Cylinders["MM346_RivetingSupportLeft"].ToBp
   END_STEP
   TRANSITION Trans36 FROM "Wedge cylinders back." TO "Support cylinders back."   // T36
      := "DevicesData".Cylinders["MM350_ShiftWedgeRight"].InBp AND "DevicesData".Cylinders["MM352_ShiftWedgeLeft"].InBp AND "DevicesData".Cylinders["MM344_RivetingSupportRight"].InBp AND "DevicesData".Cylinders["MM346_RivetingSupportLeft"].InBp;
   END_TRANSITION
   STEP "Support cylinders back.":   // S25, max time T#10S, warning time T#7S
      supervision V := #"Support cylinders back.".T > #"Support cylinders back.".T_MAX;
              S    "DevicesData".Cylinders["MM300_ShiftingSupportRight"].ToBp
              S    "DevicesData".Cylinders["MM302_ShiftingSupportLeft"].ToBp
              S    "DevicesData".Cylinders["MM340_RivetingUnitRight"].ToBp
              S    "DevicesData".Cylinders["MM342_RivetingUnitLeft"].ToBp
   END_STEP
   TRANSITION Trans40 FROM "Support cylinders back." TO "Ready for pickup by autoeject"   // T40
      := "DevicesData".Cylinders["MM300_ShiftingSupportRight"].InBp AND "DevicesData".Cylinders["MM302_ShiftingSupportLeft"].InBp AND "DevicesData".Cylinders["MM340_RivetingUnitRight"].InBp AND "DevicesData".Cylinders["MM342_RivetingUnitLeft"].InBp;
   END_TRANSITION

   // permanent post-instructions
   NETWORK 1
   TITLE = Hydraulic cylinders back
      #_w1 := #"Hydraulic cylinders back".X OR #"Hydraulic cylinders back.".X;
      IF #_w1 AND NOT "DevicesData".cupformingLeft_cylinder.Status.InBp THEN
          "DevicesData".cupformingLeft_cylinder.Status.ToBp := TRUE;
      END_IF;
      IF #_w1 AND NOT "DevicesData".cupformingRight_cylinder.Status.InBp THEN
          "DevicesData".cupformingRight_cylinder.Status.ToBp := TRUE;
      END_IF;
      IF #_w1 AND "DevicesData".cupformingLeft_cylinder.Status.InBp THEN
          "DevicesData".cupformingLeft_cylinder.Status.ToBp := FALSE;
      END_IF;
      IF #_w1 AND "DevicesData".cupformingRight_cylinder.Status.InBp THEN
          "DevicesData".cupformingRight_cylinder.Status.ToBp := FALSE;
      END_IF;
END_FUNCTION_BLOCK

FUNCTION_BLOCK "sq_manipulator"   // FB44, GRAPH
VERSION : 0.1
// stored: AcknowledgeErrorsRequired true, AutoNumber true, GraphVersion 6.0, InitialValuesAcquisition false, IsIECCheckEnabled false, LanguageInNetworks LAD, LockOperatingMode false, PermanentILProcessingInMANMode false, SetENOAutomatically false, SkipSteps false, UDAEnableTagReadback false, WithAlarmHandling true
   // inherited from GRAPH_BASE
   VAR
      OFF_SQ_BASE : Bool;
   END_VAR
   VAR_INPUT
      OFF_SQ { ExternalAccessible := 'False'; ExternalVisible := 'False'; ExternalWritable := 'False'} : Bool := false;   // Turn sequence off
      INIT_SQ { ExternalAccessible := 'False'; ExternalVisible := 'False'; ExternalWritable := 'False'} : Bool := false;   // Set sequence to initial state
      ACK_EF { ExternalAccessible := 'False'; ExternalVisible := 'False'; ExternalWritable := 'False'} : Bool := false;   // Acknowledge all errors and faults
      S_PREV { ExternalAccessible := 'False'; ExternalVisible := 'False'; ExternalWritable := 'False'} : Bool := false;   // Output previous step in parameter S_NO
      S_NEXT { ExternalAccessible := 'False'; ExternalVisible := 'False'; ExternalWritable := 'False'} : Bool := false;   // Indicate next step in parameter S_NO
      SW_AUTO { ExternalAccessible := 'False'; ExternalVisible := 'False'; ExternalWritable := 'False'} : Bool := false;   // Automatic mode
      SW_TAP { ExternalAccessible := 'False'; ExternalVisible := 'False'; ExternalWritable := 'False'} : Bool := false;   // Semiautomatic/switch with transition
      SW_TOP { ExternalAccessible := 'False'; ExternalVisible := 'False'; ExternalWritable := 'False'} : Bool := false;   // Semiautomatic/ignore transition
      SW_MAN { ExternalAccessible := 'False'; ExternalVisible := 'False'; ExternalWritable := 'False'} : Bool := false;   // Manual mode
      S_SEL { ExternalAccessible := 'False'; ExternalVisible := 'False'; ExternalWritable := 'False'} : Int := 0;   // Select step to be output to S_NO
      S_ON { ExternalAccessible := 'False'; ExternalVisible := 'False'; ExternalWritable := 'False'} : Bool := false;   // Activate step indicated in S_NO
      S_OFF { ExternalAccessible := 'False'; ExternalVisible := 'False'; ExternalWritable := 'False'} : Bool := false;   // Deactivate step indicated S_NO
      T_PUSH { ExternalAccessible := 'False'; ExternalVisible := 'False'; ExternalWritable := 'False'} : Bool := false;   // Enable transition to switch in semi automatic mode
   END_VAR
   VAR_OUTPUT
      S_NO { ExternalAccessible := 'False'; ExternalVisible := 'False'; ExternalWritable := 'False'} : Int := 0;   // Step number
      S_MORE { ExternalAccessible := 'False'; ExternalVisible := 'False'; ExternalWritable := 'False'} : Bool := false;   // More steps are available and can be shown in S_NO
      S_ACTIVE { ExternalAccessible := 'False'; ExternalVisible := 'False'; ExternalWritable := 'False'} : Bool := false;   // Step indicated in S_NO is active
      ERR_FLT { ExternalAccessible := 'False'; ExternalVisible := 'False'; ExternalWritable := 'False'} : Bool := false;   // Interlock or supervision group error
      AUTO_ON { ExternalAccessible := 'False'; ExternalVisible := 'False'; ExternalWritable := 'False'} : Bool := false;   // Automatic mode is active
      TAP_ON { ExternalAccessible := 'False'; ExternalVisible := 'False'; ExternalWritable := 'False'} : Bool := false;   // Semiautomatic mode/step with transition enabled
      TOP_ON { ExternalAccessible := 'False'; ExternalVisible := 'False'; ExternalWritable := 'False'} : Bool := false;   // Semiautomatic mode/ignore transition enabled
      MAN_ON { ExternalAccessible := 'False'; ExternalVisible := 'False'; ExternalWritable := 'False'} : Bool := false;   // Manual mode is active
   END_VAR
   VAR
      dummy : Bool;
      start : Bool;
      base : Bool;
      IEC_Timer_0_Instance { S7_SetPoint := 'True'} : TON_TIME;
      IEC_Timer_0_Instance_1 { S7_SetPoint := 'True'} : TON_TIME;
      IEC_Timer_0_Instance_2 { S7_SetPoint := 'True'} : TON_TIME;
   END_VAR
BEGIN
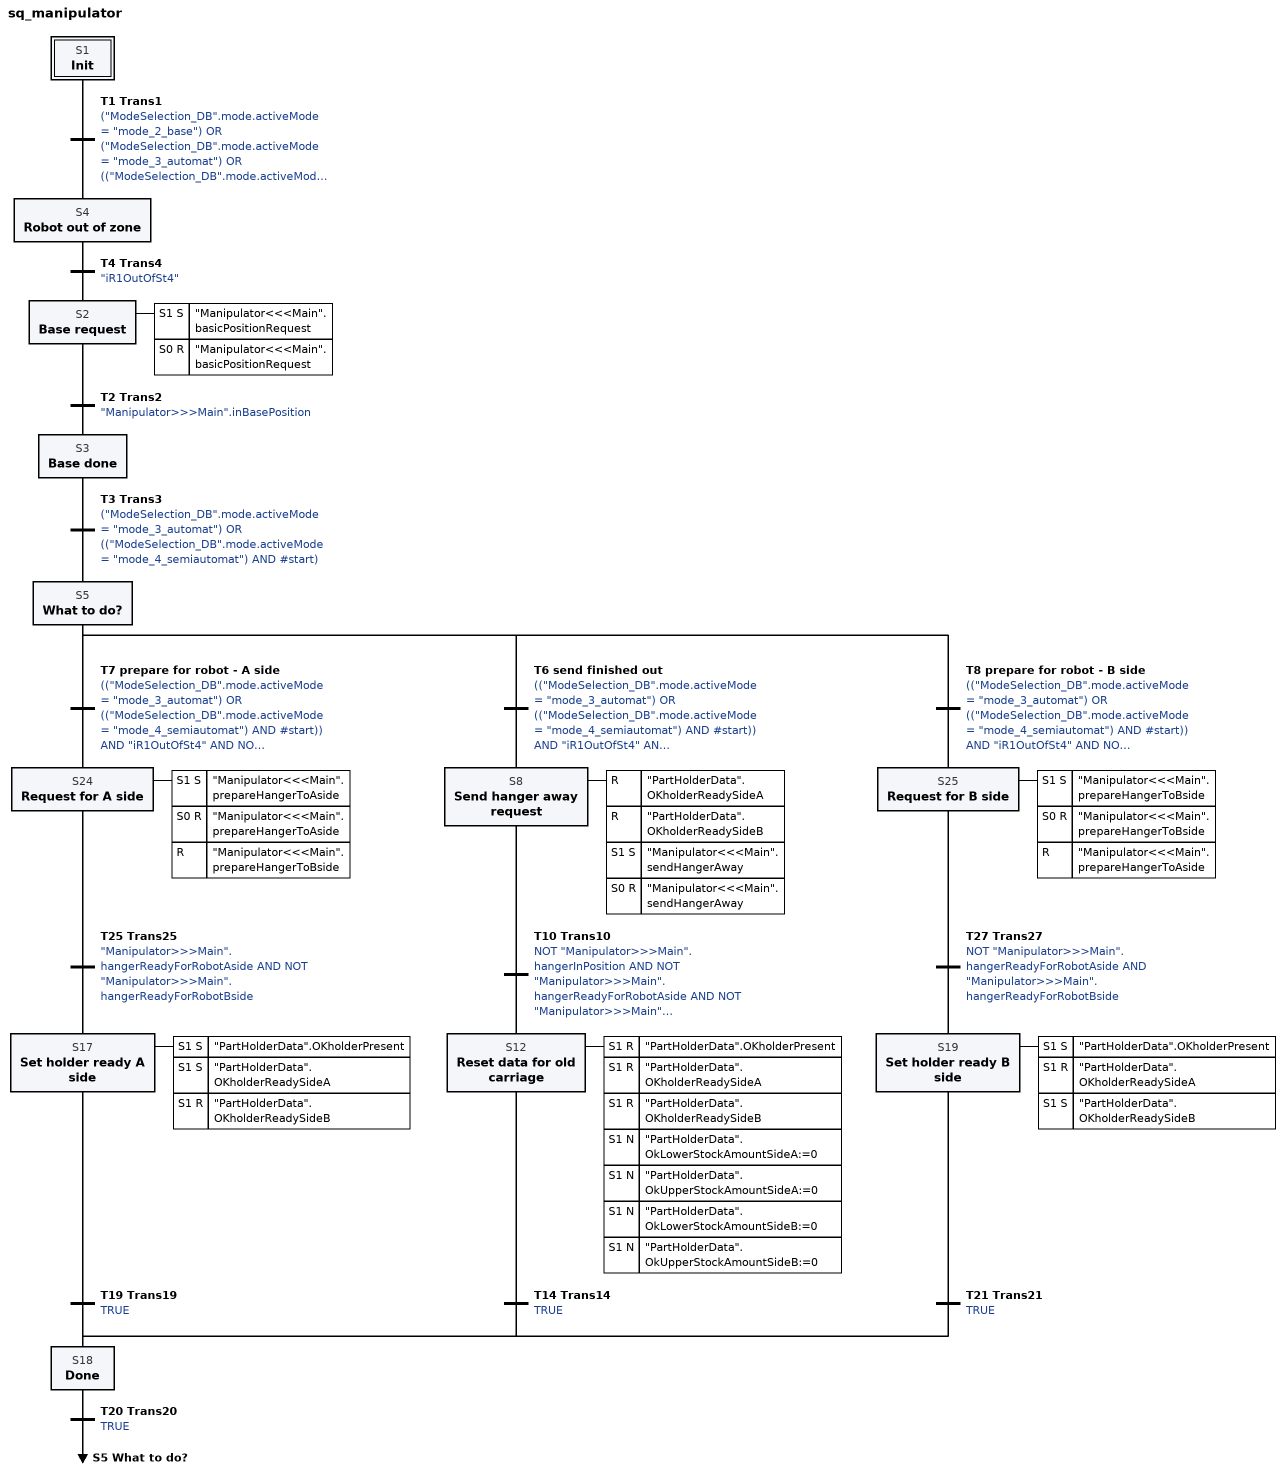
   // permanent pre-instructions
   NETWORK 1
   TITLE = base
      #base := #"Base done".X;

   // sequencer 1
   INITIAL_STEP Init:   // S1, max time T#10S, warning time T#7S
   END_STEP
   TRANSITION Trans1 FROM Init TO "Robot out of zone"   // T1
      := ("ModeSelection_DB".mode.activeMode = "mode_2_base") OR ("ModeSelection_DB".mode.activeMode = "mode_3_automat") OR (("ModeSelection_DB".mode.activeMode = "mode_4_semiautomat") AND #start);
   END_TRANSITION
   STEP "Base request":   // S2, max time T#10S, warning time T#7S
          S1  S    "Manipulator<<<Main".basicPositionRequest
          S0  R    "Manipulator<<<Main".basicPositionRequest
   END_STEP
   TRANSITION Trans2 FROM "Base request" TO "Base done"   // T2
      := "Manipulator>>>Main".inBasePosition;
   END_TRANSITION
   STEP "Base done":   // S3, max time T#10S, warning time T#7S
   END_STEP
   TRANSITION Trans3 FROM "Base done" TO "What to do?"   // T3
      := ("ModeSelection_DB".mode.activeMode = "mode_3_automat") OR (("ModeSelection_DB".mode.activeMode = "mode_4_semiautomat") AND #start);
   END_TRANSITION
   STEP "Robot out of zone":   // S4, max time T#10S, warning time T#7S
      supervision V := (#"Robot out of zone".T > #"Robot out of zone".T_MAX) AND (T#0MS > #"Robot out of zone".T_MAX);
   END_STEP
   TRANSITION Trans4 FROM "Robot out of zone" TO "Base request"   // T4
      := "iR1OutOfSt4";
   END_TRANSITION
   STEP "What to do?":   // S5, max time T#10S, warning time T#7S
   END_STEP
   TRANSITION "prepare for robot - A side" FROM "What to do?" TO "Request for A side"   // T7
      := (("ModeSelection_DB".mode.activeMode = "mode_3_automat") OR (("ModeSelection_DB".mode.activeMode = "mode_4_semiautomat") AND #start)) AND "iR1OutOfSt4" AND NOT "PartHolderData".OKholderReadySideA AND (("PartHolderData".OkLowerStockAmountSideA < "StationParameters".OKLowerStockSize) OR ("PartHolderData".OkUpperStockAmountSideA < "StationParameters".OKUpperStockSize));
   END_TRANSITION
   TRANSITION "send finished out" FROM "What to do?" TO "Send hanger away request"   // T6
      := (("ModeSelection_DB".mode.activeMode = "mode_3_automat") OR (("ModeSelection_DB".mode.activeMode = "mode_4_semiautomat") AND #start)) AND "iR1OutOfSt4" AND "PartHolderData".OKholderPresent AND ("PartHolderData".OkLowerStockAmountSideA >= "StationParameters".OKLowerStockSize) AND ("PartHolderData".OkUpperStockAmountSideA >= "StationParameters".OKUpperStockSize) AND ("PartHolderData".OkLowerStockAmountSideB >= "StationParameters".OKLowerStockSize) AND ("PartHolderData".OkUpperStockAmountSideB >= "StationParameters".OKUpperStockSize) AND NOT "sq_robot_"."Dropoff part to manipulator level1".X AND NOT "sq_robot_"."Dropoff part to manipulator level2".X;
   END_TRANSITION
   TRANSITION "prepare for robot - B side" FROM "What to do?" TO "Request for B side"   // T8
      := (("ModeSelection_DB".mode.activeMode = "mode_3_automat") OR (("ModeSelection_DB".mode.activeMode = "mode_4_semiautomat") AND #start)) AND "iR1OutOfSt4" AND NOT "PartHolderData".OKholderReadySideB AND (("PartHolderData".OkLowerStockAmountSideB < "StationParameters".OKLowerStockSize) OR ("PartHolderData".OkUpperStockAmountSideB < "StationParameters".OKUpperStockSize)) AND ("PartHolderData".OkLowerStockAmountSideA >= "StationParameters".OKLowerStockSize) AND ("PartHolderData".OkUpperStockAmountSideA >= "StationParameters".OKUpperStockSize);
   END_TRANSITION
   STEP "Request for B side":   // S25, max time T#30S, warning time T#7S
      supervision V := (#"Request for B side".T > #"Request for B side".T_MAX) AND (T#0MS > #"Request for B side".T_MAX);
          S1  S    "Manipulator<<<Main".prepareHangerToBside
          S0  R    "Manipulator<<<Main".prepareHangerToBside
              R    "Manipulator<<<Main".prepareHangerToAside
   END_STEP
   TRANSITION Trans27 FROM "Request for B side" TO "Set holder ready B side"   // T27
      := NOT "Manipulator>>>Main".hangerReadyForRobotAside AND "Manipulator>>>Main".hangerReadyForRobotBside;
   END_TRANSITION
   STEP "Set holder ready A side":   // S17, max time T#10S, warning time T#7S
          S1  S    "PartHolderData".OKholderPresent
          S1  S    "PartHolderData".OKholderReadySideA
          S1  R    "PartHolderData".OKholderReadySideB
   END_STEP
   TRANSITION Trans19 FROM "Set holder ready A side" TO Done   // T19
      := TRUE;
   END_TRANSITION
   STEP Done:   // S18, max time T#10S, warning time T#7S
   END_STEP
   TRANSITION Trans20 FROM Done TO "What to do?"   // T20, jump
      := TRUE;
   END_TRANSITION
   STEP "Send hanger away request":   // S8, max time T#10S, warning time T#7S
              R    "PartHolderData".OKholderReadySideA
              R    "PartHolderData".OKholderReadySideB
          S1  S    "Manipulator<<<Main".sendHangerAway
          S0  R    "Manipulator<<<Main".sendHangerAway
   END_STEP
   TRANSITION Trans10 FROM "Send hanger away request" TO "Reset data for old carriage"   // T10
      := NOT "Manipulator>>>Main".hangerInPosition AND NOT "Manipulator>>>Main".hangerReadyForRobotAside AND NOT "Manipulator>>>Main".hangerReadyForRobotBside;
   END_TRANSITION
   STEP "Set holder ready B side":   // S19, max time T#10S, warning time T#7S
          S1  S    "PartHolderData".OKholderPresent
          S1  R    "PartHolderData".OKholderReadySideA
          S1  S    "PartHolderData".OKholderReadySideB
   END_STEP
   TRANSITION Trans21 FROM "Set holder ready B side" TO Done   // T21
      := TRUE;
   END_TRANSITION
   STEP "Reset data for old carriage":   // S12, max time T#10S, warning time T#7S
          S1  R    "PartHolderData".OKholderPresent
          S1  R    "PartHolderData".OKholderReadySideA
          S1  R    "PartHolderData".OKholderReadySideB
          S1  N    "PartHolderData".OkLowerStockAmountSideA:=0
          S1  N    "PartHolderData".OkUpperStockAmountSideA:=0
          S1  N    "PartHolderData".OkLowerStockAmountSideB:=0
          S1  N    "PartHolderData".OkUpperStockAmountSideB:=0
   END_STEP
   TRANSITION Trans14 FROM "Reset data for old carriage" TO Done   // T14
      := TRUE;
   END_TRANSITION
   STEP "Request for A side":   // S24, max time T#30S, warning time T#7S
      supervision V := (#"Request for A side".T > #"Request for A side".T_MAX) AND (T#0MS > #"Request for A side".T_MAX);
          S1  S    "Manipulator<<<Main".prepareHangerToAside
          S0  R    "Manipulator<<<Main".prepareHangerToAside
              R    "Manipulator<<<Main".prepareHangerToBside
   END_STEP
   TRANSITION Trans25 FROM "Request for A side" TO "Set holder ready A side"   // T25
      := "Manipulator>>>Main".hangerReadyForRobotAside AND NOT "Manipulator>>>Main".hangerReadyForRobotBside;
   END_TRANSITION
END_FUNCTION_BLOCK

FUNCTION_BLOCK "sq_robot"   // FB42, GRAPH
VERSION : 0.1
// stored: AcknowledgeErrorsRequired true, AutoNumber true, GraphVersion 6.0, InitialValuesAcquisition false, IsIECCheckEnabled false, LanguageInNetworks LAD, LockOperatingMode false, PermanentILProcessingInMANMode false, SetENOAutomatically false, SkipSteps false, UDAEnableTagReadback false, WithAlarmHandling true
   // inherited from GRAPH_BASE
   VAR
      OFF_SQ_BASE : Bool;
   END_VAR
   VAR_INPUT
      OFF_SQ { ExternalWritable := 'False'} : Bool := false;   // Turn sequence off
      INIT_SQ { ExternalWritable := 'False'} : Bool := false;   // Set sequence to initial state
      ACK_EF { ExternalWritable := 'False'} : Bool := false;   // Acknowledge all errors and faults
      S_PREV { ExternalWritable := 'False'} : Bool := false;   // Output previous step in parameter S_NO
      S_NEXT { ExternalWritable := 'False'} : Bool := false;   // Indicate next step in parameter S_NO
      SW_AUTO { ExternalWritable := 'False'} : Bool := false;   // Automatic mode
      SW_TAP { ExternalWritable := 'False'} : Bool := false;   // Semiautomatic/switch with transition
      SW_TOP { ExternalWritable := 'False'} : Bool := false;   // Semiautomatic/ignore transition
      SW_MAN { ExternalWritable := 'False'} : Bool := false;   // Manual mode
      S_SEL { ExternalWritable := 'False'} : Int := 0;   // Select step to be output to S_NO
      S_ON { ExternalWritable := 'False'} : Bool := false;   // Activate step indicated in S_NO
      S_OFF { ExternalWritable := 'False'} : Bool := false;   // Deactivate step indicated S_NO
      T_PUSH { ExternalWritable := 'False'} : Bool := false;   // Enable transition to switch in semi automatic mode
   END_VAR
   VAR_OUTPUT
      S_NO { ExternalWritable := 'False'} : Int := 0;   // Step number
      S_MORE { ExternalWritable := 'False'} : Bool := false;   // More steps are available and can be shown in S_NO
      S_ACTIVE { ExternalWritable := 'False'} : Bool := false;   // Step indicated in S_NO is active
      ERR_FLT { ExternalWritable := 'False'} : Bool := false;   // Interlock or supervision group error
      AUTO_ON { ExternalWritable := 'False'} : Bool := false;   // Automatic mode is active
      TAP_ON { ExternalWritable := 'False'} : Bool := false;   // Semiautomatic mode/step with transition enabled
      TOP_ON { ExternalWritable := 'False'} : Bool := false;   // Semiautomatic mode/ignore transition enabled
      MAN_ON { ExternalWritable := 'False'} : Bool := false;   // Manual mode is active
   END_VAR
   VAR
      dummy : Bool;
      start : Bool;
      base : Bool;
      startMastering : Bool;
      startBraketest : Bool;
      prgNrForManipulatorDropoff : Byte;
   END_VAR
   VAR CONSTANT
      jobHoming : Byte := 1;
      jobCarouselPickup : Byte := 2;
      jobJigDropoff : Byte := 3;
      jobAutoEjectPickup : Byte := 4;
      jobMastering : Byte := 10;
      jobBreaktest : Byte := 11;
      jobManipulatorDropoff1 : Byte := 21;   // top far
      jobManipulatorDropoff2 : Byte := 22;   // top middle
      jobManipulatorDropoff3 : Byte := 23;   // top near
      jobManipulatorDropoff4 : Byte := 24;   // bottom far
      jobManipulatorDropoff5 : Byte := 25;   // bottom middle
      jobManipulatorDropoff6 : Byte := 26;   // bottom near
      jobManipulatorForTesting : Byte := 30;
   END_VAR
   VAR_TEMP   // added for the SCL form of the ladder/FBD networks
      _w1 : Bool;
      _w2 : Bool;
   END_VAR
BEGIN
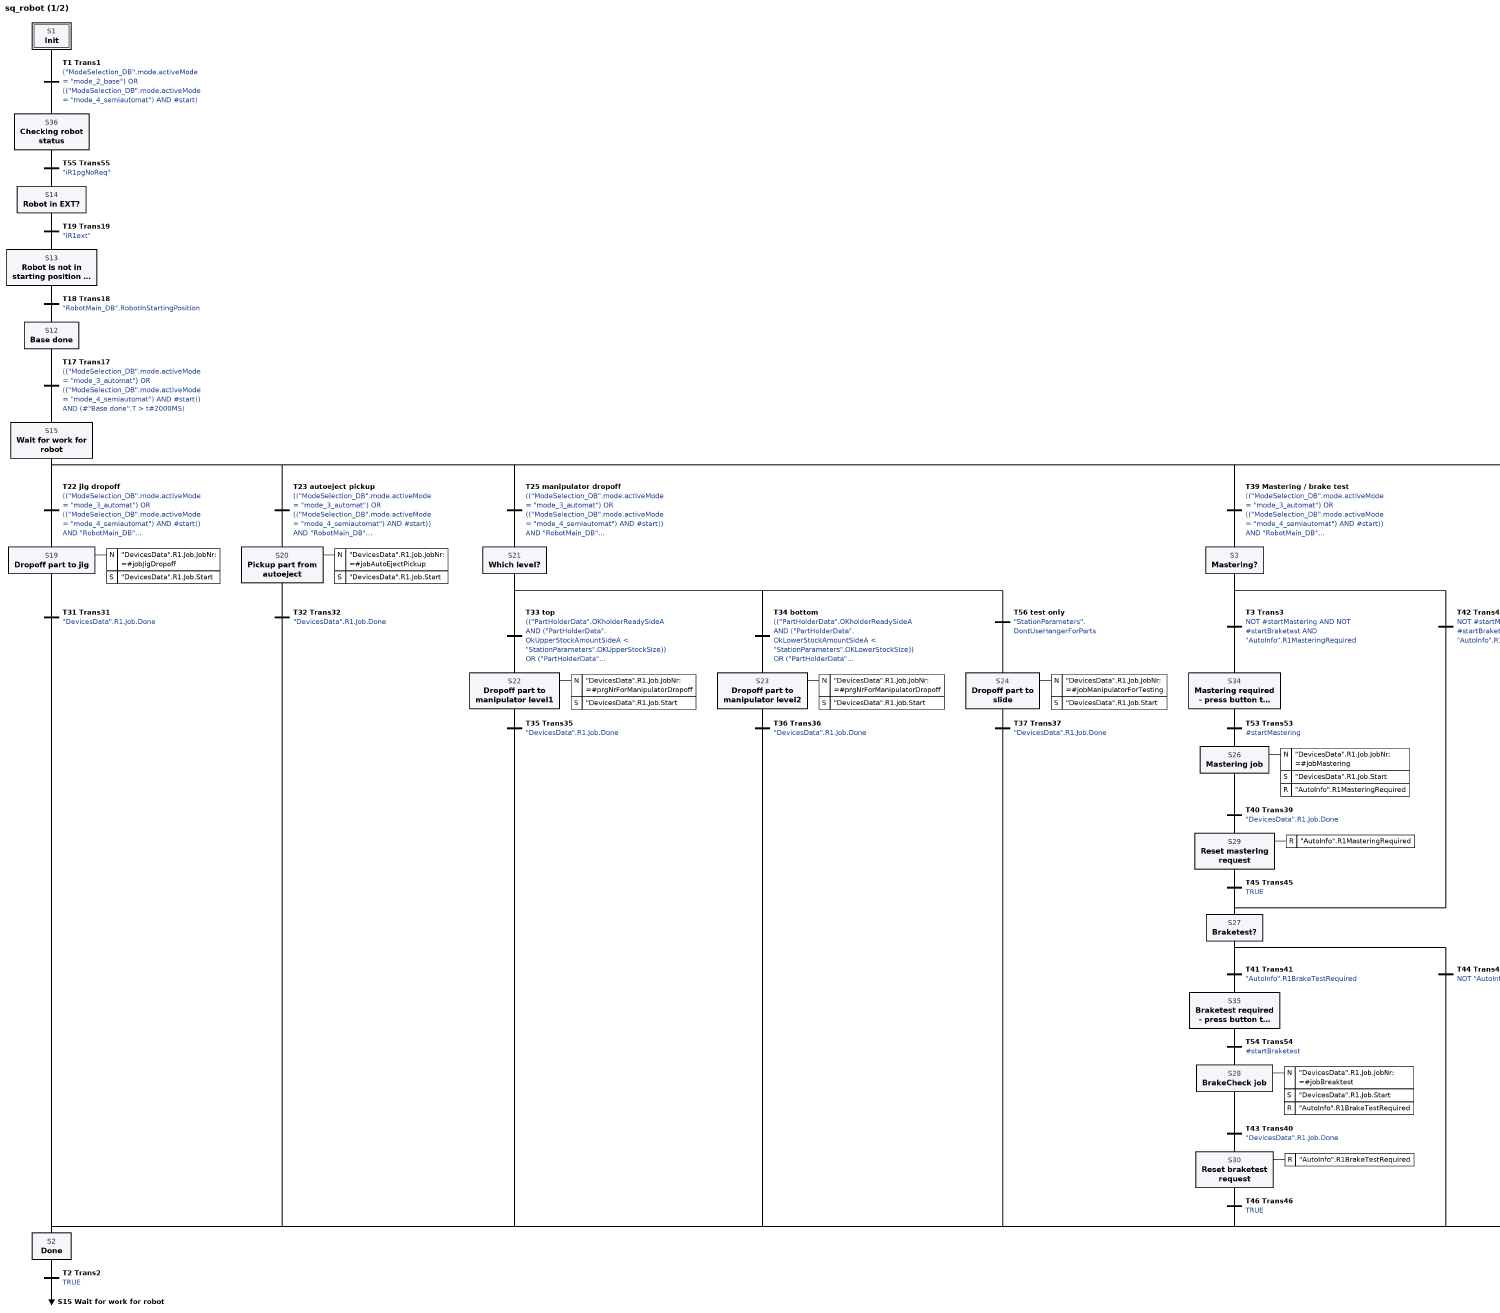
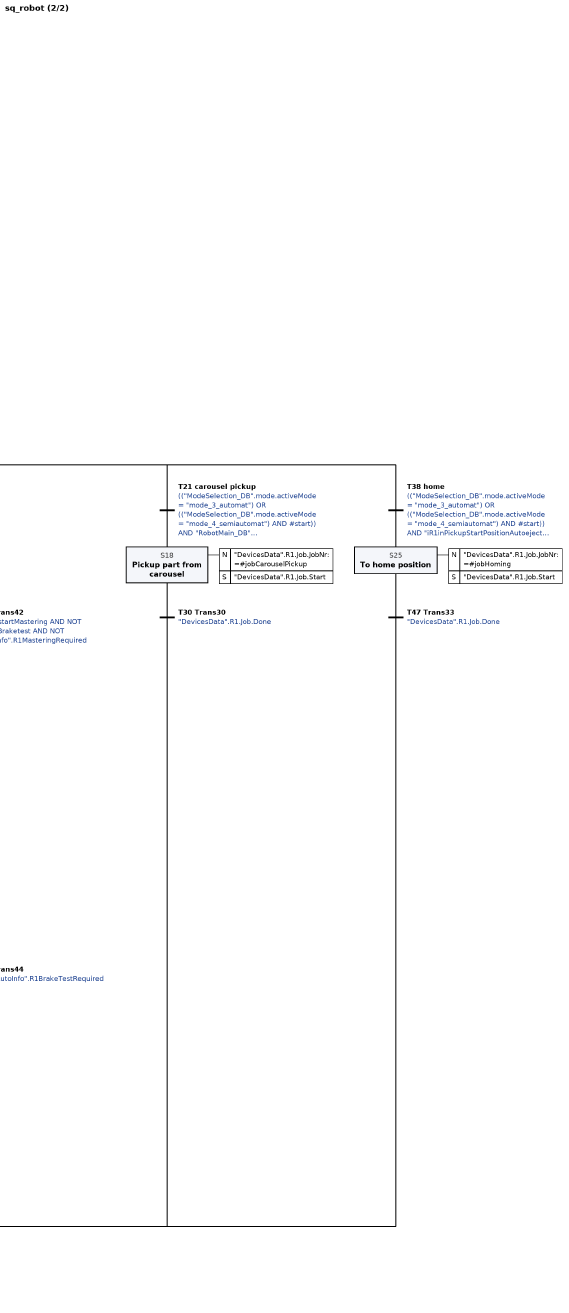
   // permanent pre-instructions
   NETWORK 1
   TITLE = prg for top level
      #_w1 := #"Dropoff part to manipulator level1".S1 AND "PartHolderData".OKholderReadySideA AND NOT "PartHolderData".OKholderReadySideB;
      IF #_w1 AND ("PartHolderData".OkUpperStockAmountSideA = 0) THEN
          #prgNrForManipulatorDropoff := #jobManipulatorDropoff1;
      END_IF;
      IF #_w1 AND ("PartHolderData".OkUpperStockAmountSideA = 1) THEN
          #prgNrForManipulatorDropoff := #jobManipulatorDropoff2;
      END_IF;
      IF #_w1 AND ("PartHolderData".OkUpperStockAmountSideA = 2) THEN
          #prgNrForManipulatorDropoff := #jobManipulatorDropoff3;
      END_IF;
      #_w2 := #"Dropoff part to manipulator level1".S1 AND NOT "PartHolderData".OKholderReadySideA AND "PartHolderData".OKholderReadySideB;
      IF #_w2 AND ("PartHolderData".OkUpperStockAmountSideB = 0) THEN
          #prgNrForManipulatorDropoff := #jobManipulatorDropoff1;
      END_IF;
      IF #_w2 AND ("PartHolderData".OkUpperStockAmountSideB = 1) THEN
          #prgNrForManipulatorDropoff := #jobManipulatorDropoff2;
      END_IF;
      IF #_w2 AND ("PartHolderData".OkUpperStockAmountSideB = 2) THEN
          #prgNrForManipulatorDropoff := #jobManipulatorDropoff3;
      END_IF;
   NETWORK 2
   TITLE = prg for bottom level
      #_w1 := #"Dropoff part to manipulator level2".S1 AND "PartHolderData".OKholderReadySideA AND NOT "PartHolderData".OKholderReadySideB;
      IF #_w1 AND ("PartHolderData".OkLowerStockAmountSideA = 0) THEN
          #prgNrForManipulatorDropoff := #jobManipulatorDropoff4;
      END_IF;
      IF #_w1 AND ("PartHolderData".OkLowerStockAmountSideA = 1) THEN
          #prgNrForManipulatorDropoff := #jobManipulatorDropoff5;
      END_IF;
      IF #_w1 AND ("PartHolderData".OkLowerStockAmountSideA = 2) THEN
          #prgNrForManipulatorDropoff := #jobManipulatorDropoff6;
      END_IF;
      #_w2 := #"Dropoff part to manipulator level2".S1 AND NOT "PartHolderData".OKholderReadySideA AND "PartHolderData".OKholderReadySideB;
      IF #_w2 AND ("PartHolderData".OkLowerStockAmountSideB = 0) THEN
          #prgNrForManipulatorDropoff := #jobManipulatorDropoff4;
      END_IF;
      IF #_w2 AND ("PartHolderData".OkLowerStockAmountSideB = 1) THEN
          #prgNrForManipulatorDropoff := #jobManipulatorDropoff5;
      END_IF;
      IF #_w2 AND ("PartHolderData".OkLowerStockAmountSideB = 2) THEN
          #prgNrForManipulatorDropoff := #jobManipulatorDropoff6;
      END_IF;
   NETWORK 3
      #base := "RobotMain_DB".RobotInStartingPosition AND "iR1ext";
   NETWORK 4
   TITLE = job start init
      "DevicesData".R1.Job.Start := FALSE;
   NETWORK 5
      "qR1_ST3free" := "sq_fitting_station_st3".base;

   // sequencer 1
   INITIAL_STEP Init:   // S1, max time T#10S, warning time T#7S
   END_STEP
   TRANSITION Trans1 FROM Init TO "Checking robot status"   // T1
      := ("ModeSelection_DB".mode.activeMode = "mode_2_base") OR (("ModeSelection_DB".mode.activeMode = "mode_4_semiautomat") AND #start);
   END_TRANSITION
   STEP Done:   // S2, max time T#10S, warning time T#7S
   END_STEP
   TRANSITION Trans2 FROM Done TO "Wait for work for robot"   // T2, jump
      := TRUE;
   END_TRANSITION
   STEP "Base done":   // S12, max time T#10S, warning time T#7S
   END_STEP
   TRANSITION Trans17 FROM "Base done" TO "Wait for work for robot"   // T17
      := (("ModeSelection_DB".mode.activeMode = "mode_3_automat") OR (("ModeSelection_DB".mode.activeMode = "mode_4_semiautomat") AND #start)) AND (#"Base done".T > t#2000MS);
   END_TRANSITION
   STEP "Robot is not in starting position - move it to home manualy":   // S13, max time T#1S, warning time T#7S
      supervision V := #"Robot is not in starting position - move it to home manualy".T > #"Robot is not in starting position - move it to home manualy".T_MAX;
   END_STEP
   TRANSITION Trans18 FROM "Robot is not in starting position - move it to home manualy" TO "Base done"   // T18
      := "RobotMain_DB".RobotInStartingPosition;
   END_TRANSITION
   STEP "Robot in EXT?":   // S14, max time T#10S, warning time T#7S
      supervision V := #"Robot in EXT?".T > #"Robot in EXT?".T_MAX;
   END_STEP
   TRANSITION Trans19 FROM "Robot in EXT?" TO "Robot is not in starting position - move it to home manualy"   // T19
      := "iR1ext";
   END_TRANSITION
   STEP "Wait for work for robot":   // S15, max time T#10S, warning time T#7S
   END_STEP
   TRANSITION "jig dropoff" FROM "Wait for work for robot" TO "Dropoff part to jig"   // T22
      := (("ModeSelection_DB".mode.activeMode = "mode_3_automat") OR (("ModeSelection_DB".mode.activeMode = "mode_4_semiautomat") AND #start)) AND "RobotMain_DB".RobotInStartingPosition AND "sq_fitting_station_st3"."Waiting for the part to be inserted".X AND "DevicesData"."TA1-3MA".data.zones.outOfST3zone AND NOT "AutoPositions".St3_Fitting.PartPresent AND NOT "i3partPresent" AND "AutoPositions".R1_Gripper.PartPresent AND "iR1tubePresentFront" AND "iR1tubePresentRear" AND NOT "AutoPositions".R1_Gripper.StFinished[3] AND NOT "AutoPositions".R1_Gripper.PartNOK AND "sq_fitting_station_st3".base;
   END_TRANSITION
   TRANSITION "autoeject pickup" FROM "Wait for work for robot" TO "Pickup part from autoeject"   // T23
      := (("ModeSelection_DB".mode.activeMode = "mode_3_automat") OR (("ModeSelection_DB".mode.activeMode = "mode_4_semiautomat") AND #start)) AND "RobotMain_DB".RobotInStartingPosition AND "DevicesData"."TA1-3MA".data.zones.outOfOKposZone AND ((NOT "AutoInfo".EndProduction AND "AutoPositions".St3_Fitting.PartPresent) OR "AutoInfo".EndProduction) AND ("i4partPresent" OR "StationParameters".GhostMode) AND NOT "AutoPositions".R1_Gripper.PartPresent AND NOT "iR1tubePresentFront" AND NOT "iR1tubePresentRear" AND "AutoPositions".St4_OKposition.PartPresent;
   END_TRANSITION
   TRANSITION "manipulator dropoff" FROM "Wait for work for robot" TO "Which level?"   // T25
      := (("ModeSelection_DB".mode.activeMode = "mode_3_automat") OR (("ModeSelection_DB".mode.activeMode = "mode_4_semiautomat") AND #start)) AND "RobotMain_DB".RobotInStartingPosition AND (("PartHolderData".OKholderReadySideA AND (("PartHolderData".OkLowerStockAmountSideA < "StationParameters".OKLowerStockSize) OR ("PartHolderData".OkUpperStockAmountSideA < "StationParameters".OKUpperStockSize))) OR ("PartHolderData".OKholderReadySideB AND (("PartHolderData".OkLowerStockAmountSideB < "StationParameters".OKLowerStockSize) OR ("PartHolderData".OkUpperStockAmountSideB < "StationParameters".OKUpperStockSize)))) AND "AutoPositions".R1_Gripper.PartPresent AND "iR1tubePresentFront" AND "iR1tubePresentRear" AND "AutoPositions".R1_Gripper.StFinished[3] AND NOT "AutoPositions".R1_Gripper.PartNOK;
   END_TRANSITION
   TRANSITION "Mastering / brake test" FROM "Wait for work for robot" TO "Mastering?"   // T39
      := (("ModeSelection_DB".mode.activeMode = "mode_3_automat") OR (("ModeSelection_DB".mode.activeMode = "mode_4_semiautomat") AND #start)) AND "RobotMain_DB".RobotInStartingPosition AND "DevicesData"."TA1-3MA".data.zones.outOfST3zone AND NOT "AutoPositions".R1_Gripper.PartPresent AND NOT "iR1tubePresentFront" AND NOT "iR1tubePresentRear" AND ("AutoInfo".R1MasteringRequired OR "AutoInfo".R1BrakeTestRequired);
   END_TRANSITION
   TRANSITION "carousel pickup" FROM "Wait for work for robot" TO "Pickup part from carousel"   // T21
      := (("ModeSelection_DB".mode.activeMode = "mode_3_automat") OR (("ModeSelection_DB".mode.activeMode = "mode_4_semiautomat") AND #start)) AND "RobotMain_DB".RobotInStartingPosition AND "sq_carousel_unloading_st2"."Wait for robot to remove part".X AND "AutoPositions".St2_Table2.PartPresent AND (NOT "AutoPositions".St3_Fitting.PartPresent OR NOT "AutoPositions".St4_OKposition.PartPresent) AND NOT "AutoPositions".St2_Table2.PartNOK AND NOT "AutoPositions".R1_Gripper.PartPresent AND NOT "iR1tubePresentFront" AND NOT "iR1tubePresentRear" AND "iTableInPosition" AND "iTurnTableIndexerInPosition";
   END_TRANSITION
   TRANSITION home FROM "Wait for work for robot" TO "To home position"   // T38
      := (("ModeSelection_DB".mode.activeMode = "mode_3_automat") OR (("ModeSelection_DB".mode.activeMode = "mode_4_semiautomat") AND #start)) AND "iR1inPickupStartPositionAutoeject" AND "AutoInfo".EndProduction AND NOT "AutoPositions".St2_Table2.PartPresent AND "AutoPositions".St3_Fitting.PartPresent AND "i3partPresent" AND NOT "AutoPositions".St4_OKposition.PartPresent AND NOT "i4partPresent";
   END_TRANSITION
   STEP "Mastering job":   // S26, max time T#50S, warning time T#7S
      supervision V := #"Mastering job".T > #"Mastering job".T_MAX;
              N    "DevicesData".R1.Job.JobNr:=#jobMastering
              S    "DevicesData".R1.Job.Start
              R    "AutoInfo".R1MasteringRequired
   END_STEP
   TRANSITION Trans39 FROM "Mastering job" TO "Reset mastering request"   // T40
      := "DevicesData".R1.Job.Done;
   END_TRANSITION
   STEP "Dropoff part to jig":   // S19, max time T#30S, warning time T#7S
      supervision V := #"Dropoff part to jig".T > #"Dropoff part to jig".T_MAX;
              N    "DevicesData".R1.Job.JobNr:=#jobJigDropoff
              S    "DevicesData".R1.Job.Start
   END_STEP
   TRANSITION Trans31 FROM "Dropoff part to jig" TO Done   // T31
      := "DevicesData".R1.Job.Done;
   END_TRANSITION
   STEP "Pickup part from autoeject":   // S20, max time T#30S, warning time T#7S
      supervision V := #"Pickup part from autoeject".T > #"Pickup part from autoeject".T_MAX;
              N    "DevicesData".R1.Job.JobNr:=#jobAutoEjectPickup
              S    "DevicesData".R1.Job.Start
   END_STEP
   TRANSITION Trans32 FROM "Pickup part from autoeject" TO Done   // T32
      := "DevicesData".R1.Job.Done;
   END_TRANSITION
   STEP "Which level?":   // S21, max time T#10S, warning time T#7S
   END_STEP
   TRANSITION top FROM "Which level?" TO "Dropoff part to manipulator level1"   // T33
      := (("PartHolderData".OKholderReadySideA AND ("PartHolderData".OkUpperStockAmountSideA < "StationParameters".OKUpperStockSize)) OR ("PartHolderData".OKholderReadySideB AND ("PartHolderData".OkUpperStockAmountSideB < "StationParameters".OKUpperStockSize))) AND NOT "StationParameters".DontUseHangerForParts;
   END_TRANSITION
   TRANSITION bottom FROM "Which level?" TO "Dropoff part to manipulator level2"   // T34
      := (("PartHolderData".OKholderReadySideA AND ("PartHolderData".OkLowerStockAmountSideA < "StationParameters".OKLowerStockSize)) OR ("PartHolderData".OKholderReadySideB AND ("PartHolderData".OkLowerStockAmountSideB < "StationParameters".OKLowerStockSize))) AND NOT "StationParameters".DontUseHangerForParts;
   END_TRANSITION
   TRANSITION "test only" FROM "Which level?" TO "Dropoff part to slide"   // T56
      := "StationParameters".DontUseHangerForParts;
   END_TRANSITION
   STEP "Dropoff part to manipulator level1":   // S22, max time T#30S, warning time T#7S
      supervision V := (#"Dropoff part to manipulator level1".T > #"Dropoff part to manipulator level1".T_MAX) AND (#"Dropoff part to manipulator level1".T > T#60S);
              N    "DevicesData".R1.Job.JobNr:=#prgNrForManipulatorDropoff
              S    "DevicesData".R1.Job.Start
   END_STEP
   TRANSITION Trans35 FROM "Dropoff part to manipulator level1" TO Done   // T35
      := "DevicesData".R1.Job.Done;
   END_TRANSITION
   STEP "Dropoff part to manipulator level2":   // S23, max time T#30S, warning time T#7S
      supervision V := #"Dropoff part to manipulator level2".T > #"Dropoff part to manipulator level2".T_MAX;
              N    "DevicesData".R1.Job.JobNr:=#prgNrForManipulatorDropoff
              S    "DevicesData".R1.Job.Start
   END_STEP
   TRANSITION Trans36 FROM "Dropoff part to manipulator level2" TO Done   // T36
      := "DevicesData".R1.Job.Done;
   END_TRANSITION
   STEP "Mastering?":   // S3, max time T#10S, warning time T#7S
   END_STEP
   TRANSITION Trans3 FROM "Mastering?" TO "Mastering required - press button to start"   // T3
      := NOT #startMastering AND NOT #startBraketest AND "AutoInfo".R1MasteringRequired;
   END_TRANSITION
   TRANSITION Trans42 FROM "Mastering?" TO "Braketest?"   // T42
      := NOT #startMastering AND NOT #startBraketest AND NOT "AutoInfo".R1MasteringRequired;
   END_TRANSITION
   STEP "Pickup part from carousel":   // S18, max time T#30S, warning time T#7S
      supervision V := #"Pickup part from carousel".T > #"Pickup part from carousel".T_MAX;
              N    "DevicesData".R1.Job.JobNr:=#jobCarouselPickup
              S    "DevicesData".R1.Job.Start
   END_STEP
   TRANSITION Trans30 FROM "Pickup part from carousel" TO Done   // T30
      := "DevicesData".R1.Job.Done;
   END_TRANSITION
   STEP "Braketest?":   // S27, max time T#10S, warning time T#7S
   END_STEP
   TRANSITION Trans41 FROM "Braketest?" TO "Braketest required - press button to start"   // T41
      := "AutoInfo".R1BrakeTestRequired;
   END_TRANSITION
   TRANSITION Trans44 FROM "Braketest?" TO Done   // T44
      := NOT "AutoInfo".R1BrakeTestRequired;
   END_TRANSITION
   STEP "BrakeCheck job":   // S28, max time T#60S, warning time T#7S
      supervision V := #"BrakeCheck job".T > #"BrakeCheck job".T_MAX;
              N    "DevicesData".R1.Job.JobNr:=#jobBreaktest
              S    "DevicesData".R1.Job.Start
              R    "AutoInfo".R1BrakeTestRequired
   END_STEP
   TRANSITION Trans40 FROM "BrakeCheck job" TO "Reset braketest request"   // T43
      := "DevicesData".R1.Job.Done;
   END_TRANSITION
   STEP "Reset mastering request":   // S29, max time T#10S, warning time T#7S
              R    "AutoInfo".R1MasteringRequired
   END_STEP
   TRANSITION Trans45 FROM "Reset mastering request" TO "Braketest?"   // T45
      := TRUE;
   END_TRANSITION
   STEP "Reset braketest request":   // S30, max time T#10S, warning time T#7S
              R    "AutoInfo".R1BrakeTestRequired
   END_STEP
   TRANSITION Trans46 FROM "Reset braketest request" TO Done   // T46
      := TRUE;
   END_TRANSITION
   STEP "Mastering required - press button to start":   // S34, max time T#10S, warning time T#7S
   END_STEP
   TRANSITION Trans53 FROM "Mastering required - press button to start" TO "Mastering job"   // T53
      := #startMastering;
   END_TRANSITION
   STEP "Braketest required - press button to start":   // S35, max time T#10S, warning time T#7S
   END_STEP
   TRANSITION Trans54 FROM "Braketest required - press button to start" TO "BrakeCheck job"   // T54
      := #startBraketest;
   END_TRANSITION
   STEP "Checking robot status":   // S36, max time T#10S, warning time T#7S
   END_STEP
   TRANSITION Trans55 FROM "Checking robot status" TO "Robot in EXT?"   // T55
      := "iR1pgNoReq";
   END_TRANSITION
   STEP "Dropoff part to slide":   // S24, max time T#40S, warning time T#7S
      supervision V := #"Dropoff part to slide".T > #"Dropoff part to slide".T_MAX;
              N    "DevicesData".R1.Job.JobNr:=#jobManipulatorForTesting
              S    "DevicesData".R1.Job.Start
   END_STEP
   TRANSITION Trans37 FROM "Dropoff part to slide" TO Done   // T37
      := "DevicesData".R1.Job.Done;
   END_TRANSITION
   STEP "To home position":   // S25, max time T#10S, warning time T#7S
      supervision V := #"To home position".T > #"To home position".T_MAX;
              N    "DevicesData".R1.Job.JobNr:=#jobHoming
              S    "DevicesData".R1.Job.Start
   END_STEP
   TRANSITION Trans33 FROM "To home position" TO Done   // T47
      := "DevicesData".R1.Job.Done;
   END_TRANSITION

   // permanent post-instructions
   NETWORK 1
      IF #startMastering THEN #startMastering := FALSE; END_IF;
      IF #startBraketest THEN #startBraketest := FALSE; END_IF;
END_FUNCTION_BLOCK

FUNCTION_BLOCK "CylinderFaceplate"   // FB31, LAD
{ S7_Optimized_Access := 'FALSE' }
AUTHOR : Bodorik
FAMILY : RIV
NAME : Cylinder
VERSION : 0.9
// stored: AutoNumber true, IsIECCheckEnabled false, SetENOAutomatically false, UDAEnableTagReadback false
   VAR_INPUT
      POWER_OK : Bool;
      CylinderNumber : Int;
      HMICommand : Int;
      BasicPositionCondition : Bool;
      WorkPositionCondition : Bool;
      BasicPositionSensor : Bool;
      WorkPositionSensor : Bool;
      TRIGGER : Bool;
      RESET : Bool;
      DELAY_BASIC : Time;
      DELAY_WORK : Time;
      DELAY_FREE : Time;
      ERROR_TIME : Time;
      ValveDelay : Time;
      iNoCollisionBasic : Bool;
      iNoCollisionWork : Bool;
      iNoCollisionFree : Bool;
   END_VAR
   VAR_OUTPUT
      VALVE_BASIC : Bool;
      VALVE_WORK : Bool;
      ERROR_BASIC : Bool;
      ERROR_WORK : Bool;
      HMIStatus : Int;
   END_VAR
   VAR_IN_OUT
      MOVE_BASIC : Bool;
      MOVE_WORK : Bool;
      MOVE_FREE : Bool;
      CylinderOperation : "UDT_Cylinder";
   END_VAR
   VAR DB_SPECIFIC
      "4l+Started" : Bool;
      InitCommandBP : Bool;
      InitCommandWP : Bool;
      BasicWorkStartWP : Bool;
      BasicWorkStartBP : Bool;
      work_valve : Bool;
      basic_valve : Bool;
      free_valve : Bool;
      baspos_error : TON_TIME;
      workpos_error { S7_SetPoint := 'True'} : TON_TIME;
      baspos_delay { S7_SetPoint := 'True'} : TON_TIME;
      workpos_delay { S7_SetPoint := 'True'} : TON_TIME;
      CylinderOperationOld { S7_SetPoint := 'True'} : "UDT_Cylinder";
      IEC_Timer_0_Instance { S7_SetPoint := 'True'} : TP_TIME;
   END_VAR
   VAR
      R_TRIG_Instance { S7_SetPoint := 'True'} : R_TRIG;
   END_VAR
   VAR DB_SPECIFIC
      IEC_Timer_0_Instance_1 { S7_SetPoint := 'True'} : TP_TIME;
      IEC_Timer_0_Instance_2 { S7_SetPoint := 'True'} : TP_TIME;
      IEC_Timer_0_Instance_3 { S7_SetPoint := 'True'} : TON_TIME;
      IEC_Timer_0_Instance_4 { S7_SetPoint := 'True'} : TON_TIME;
   END_VAR
   VAR_TEMP
      et : Bool;
      comm : Int;
   END_VAR
   VAR_TEMP   // added for the SCL form of the ladder/FBD networks
      _w1 : Bool;
   END_VAR
BEGIN

REGION Network 1 (SCL): check new cylinder command
   //check if basic position req movement changed
   IF #CylinderOperation.ToBp <> #CylinderOperationOld.ToBp AND #CylinderOperation.ToBp THEN
       IF #iNoCollisionBasic OR (#BasicPositionCondition AND NOT #WorkPositionCondition) THEN
           #CylinderOperation.ToFp := false;
           #CylinderOperation.ToWp := false;
       ELSE
           #CylinderOperation.ToBp := false;
       END_IF;
   END_IF;
   //check if work position req movement changed
   IF #CylinderOperation.ToWp <> #CylinderOperationOld.ToWp AND #CylinderOperation.ToWp THEN
       IF #iNoCollisionWork OR (NOT #BasicPositionCondition AND #WorkPositionCondition) THEN
           #CylinderOperation.ToFp := false;
           #CylinderOperation.ToBp := false;
       ELSE
           #CylinderOperation.ToWp := false;
       END_IF;
   END_IF;
   //check if free position req movement changed
   IF #CylinderOperation.ToFp <> #CylinderOperationOld.ToFp AND #CylinderOperation.ToFp THEN
       IF #iNoCollisionFree THEN
           #CylinderOperation.ToBp := false;
           #CylinderOperation.ToWp := false;
       ELSE
           #CylinderOperation.ToFp := false;
       END_IF;
   END_IF;
   //store actual cylinder status to old
   #CylinderOperationOld := #CylinderOperation;
END_REGION

REGION Network 2 (SCL)
   #comm := #HMICommand - #CylinderNumber;
   #CylinderOperation.ToBp := #CylinderOperation.ToBp;
   #CylinderOperation.ToWp := #CylinderOperation.ToWp;
   #MOVE_BASIC := #MOVE_BASIC;
   #MOVE_WORK := #MOVE_WORK;


   IF (#comm = 1000 AND #iNoCollisionBasic) OR #CylinderOperation.ToBp THEN
       #CylinderOperation.ToBp := true;
       #CylinderOperation.ToWp := FALSE;
       #CylinderOperation.ToFp := FALSE;
       #MOVE_BASIC := true;
       #MOVE_FREE := false;
       #MOVE_WORK := false;
   END_IF;
   IF (#comm = 2000 AND #iNoCollisionWork) OR #CylinderOperation.ToWp THEN
       #CylinderOperation.ToWp := true;
       #CylinderOperation.ToBp := FALSE;
       #CylinderOperation.ToFp := FALSE;
       #MOVE_BASIC := false;
       #MOVE_FREE := false;
       #MOVE_WORK := TRUE;
   END_IF;
   IF (#comm = 3000 AND #iNoCollisionFree) OR #CylinderOperation.ToFp THEN
       #CylinderOperation.ToFp := true;
       #CylinderOperation.ToWp := FALSE;
       #CylinderOperation.ToBp := FALSE;
       #MOVE_BASIC := FALSE;
       #MOVE_FREE := TRUE;
       #MOVE_WORK := false;
   END_IF;

   IF #ERROR_BASIC OR #ERROR_WORK THEN
       #MOVE_BASIC := 0;
       #MOVE_WORK := 0;
       #CylinderOperation.ToBp := false;
       #CylinderOperation.ToWp := false;
   END_IF;

   IF NOT #POWER_OK THEN
       #MOVE_BASIC := false;
       #MOVE_WORK := false;
       #MOVE_FREE := TRUE;
       #CylinderOperation.ToBp := false;
       #CylinderOperation.ToWp := false;
       #CylinderOperation.ToFp := TRUE;
   END_IF;
END_REGION

REGION Network 3: Start movement to basic position
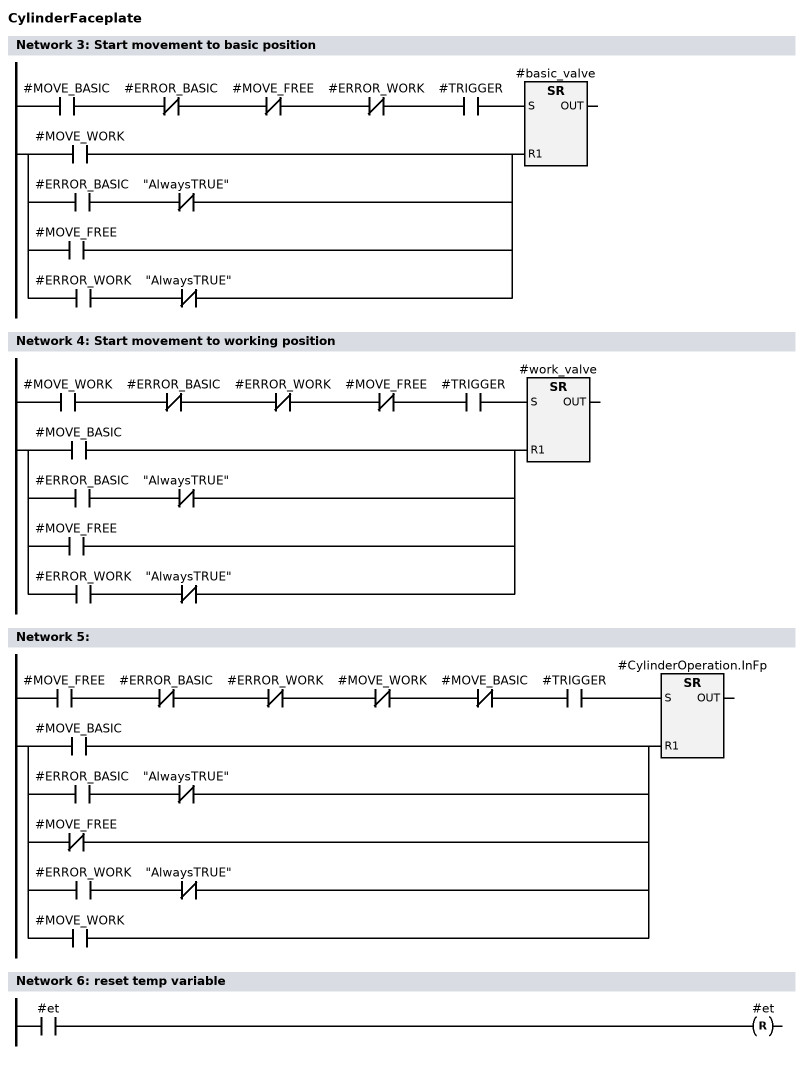
   RUNG wire#powerrail
      Contact( #MOVE_BASIC )
      I_Contact( #ERROR_BASIC )
      I_Contact( #MOVE_FREE )
      I_Contact( #ERROR_WORK )
      Contact( #TRIGGER )
      S_SR(operand := #basic_valve, r1 := wire#w1)
   END_RUNG
   RUNG wire#powerrail
      Contact( #MOVE_WORK )
   END_RUNG wire#w1
   RUNG wire#powerrail
      Contact( #ERROR_BASIC )
      I_Contact( "AlwaysTRUE" )
   END_RUNG wire#w1
   RUNG wire#powerrail
      Contact( #MOVE_FREE )
   END_RUNG wire#w1
   RUNG wire#powerrail
      Contact( #ERROR_WORK )
      I_Contact( "AlwaysTRUE" )
   END_RUNG wire#w1
   // the same network as SCL:
   IF #MOVE_BASIC AND NOT #ERROR_BASIC AND NOT #MOVE_FREE AND NOT #ERROR_WORK AND #TRIGGER THEN
       #basic_valve := TRUE;   // SR flip-flop
   END_IF;
   IF #MOVE_WORK OR (#ERROR_BASIC AND NOT "AlwaysTRUE") OR #MOVE_FREE OR (#ERROR_WORK AND NOT "AlwaysTRUE") THEN
       #basic_valve := FALSE;
   END_IF;
END_REGION

REGION Network 4: Start movement to working position
   RUNG wire#powerrail
      Contact( #MOVE_WORK )
      I_Contact( #ERROR_BASIC )
      I_Contact( #ERROR_WORK )
      I_Contact( #MOVE_FREE )
      Contact( #TRIGGER )
      S_SR(operand := #work_valve, r1 := wire#w1)
   END_RUNG
   RUNG wire#powerrail
      Contact( #MOVE_BASIC )
   END_RUNG wire#w1
   RUNG wire#powerrail
      Contact( #ERROR_BASIC )
      I_Contact( "AlwaysTRUE" )
   END_RUNG wire#w1
   RUNG wire#powerrail
      Contact( #MOVE_FREE )
   END_RUNG wire#w1
   RUNG wire#powerrail
      Contact( #ERROR_WORK )
      I_Contact( "AlwaysTRUE" )
   END_RUNG wire#w1
   // the same network as SCL:
   IF #MOVE_WORK AND NOT #ERROR_BASIC AND NOT #ERROR_WORK AND NOT #MOVE_FREE AND #TRIGGER THEN
       #work_valve := TRUE;   // SR flip-flop
   END_IF;
   IF #MOVE_BASIC OR (#ERROR_BASIC AND NOT "AlwaysTRUE") OR #MOVE_FREE OR (#ERROR_WORK AND NOT "AlwaysTRUE") THEN
       #work_valve := FALSE;
   END_IF;
END_REGION

REGION Network 5
   RUNG wire#powerrail
      Contact( #MOVE_FREE )
      I_Contact( #ERROR_BASIC )
      I_Contact( #ERROR_WORK )
      I_Contact( #MOVE_WORK )
      I_Contact( #MOVE_BASIC )
      Contact( #TRIGGER )
      S_SR(operand := #CylinderOperation.InFp, r1 := wire#w1)
   END_RUNG
   RUNG wire#powerrail
      Contact( #MOVE_BASIC )
   END_RUNG wire#w1
   RUNG wire#powerrail
      Contact( #ERROR_BASIC )
      I_Contact( "AlwaysTRUE" )
   END_RUNG wire#w1
   RUNG wire#powerrail
      I_Contact( #MOVE_FREE )
   END_RUNG wire#w1
   RUNG wire#powerrail
      Contact( #ERROR_WORK )
      I_Contact( "AlwaysTRUE" )
   END_RUNG wire#w1
   RUNG wire#powerrail
      Contact( #MOVE_WORK )
   END_RUNG wire#w1
   // the same network as SCL:
   IF #MOVE_FREE AND NOT #ERROR_BASIC AND NOT #ERROR_WORK AND NOT #MOVE_WORK AND NOT #MOVE_BASIC AND #TRIGGER THEN
       #CylinderOperation.InFp := TRUE;   // SR flip-flop
   END_IF;
   IF #MOVE_BASIC OR (#ERROR_BASIC AND NOT "AlwaysTRUE") OR NOT #MOVE_FREE OR (#ERROR_WORK AND NOT "AlwaysTRUE") OR #MOVE_WORK THEN
       #CylinderOperation.InFp := FALSE;
   END_IF;
END_REGION

REGION Network 6: reset temp variable
   RUNG wire#powerrail
      Contact( #et )
      R_Coil( #et )
   END_RUNG
   // the same network as SCL:
   IF #et THEN #et := FALSE; END_IF;
END_REGION

REGION Network 7 (FBD): Error movement to basic position
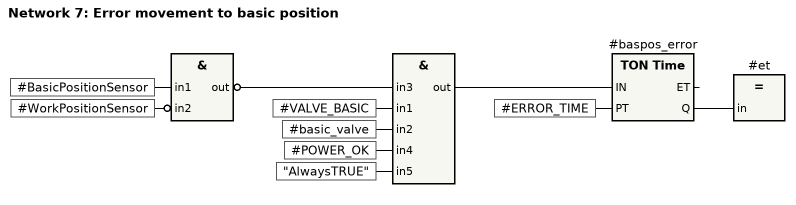
   #baspos_error(IN := NOT (#BasicPositionSensor AND NOT #WorkPositionSensor) AND #VALVE_BASIC AND #basic_valve AND #POWER_OK AND "AlwaysTRUE",   // TON
                 PT := #ERROR_TIME);
   #et := #baspos_error.Q;
END_REGION

REGION Network 8: Set basic position error
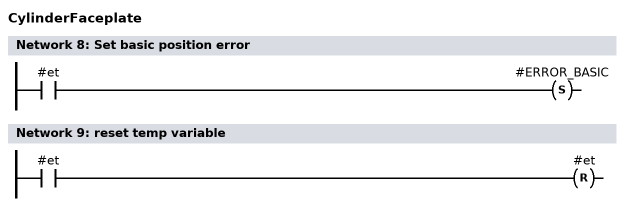
   RUNG wire#powerrail
      Contact( #et )
      S_Coil( #ERROR_BASIC )
   END_RUNG
   // the same network as SCL:
   IF #et THEN #ERROR_BASIC := TRUE; END_IF;
END_REGION

REGION Network 9: reset temp variable
   RUNG wire#powerrail
      Contact( #et )
      R_Coil( #et )
   END_RUNG
   // the same network as SCL:
   IF #et THEN #et := FALSE; END_IF;
END_REGION

REGION Network 10 (FBD): Error movement to working position
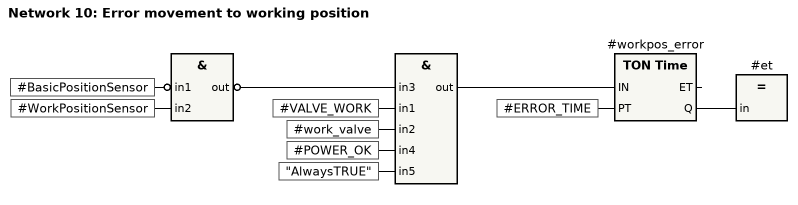
   #workpos_error(IN := NOT (NOT #BasicPositionSensor AND #WorkPositionSensor) AND #VALVE_WORK AND #work_valve AND #POWER_OK AND "AlwaysTRUE",   // TON
                  PT := #ERROR_TIME);
   #et := #workpos_error.Q;
END_REGION

REGION Network 11: Set working position error
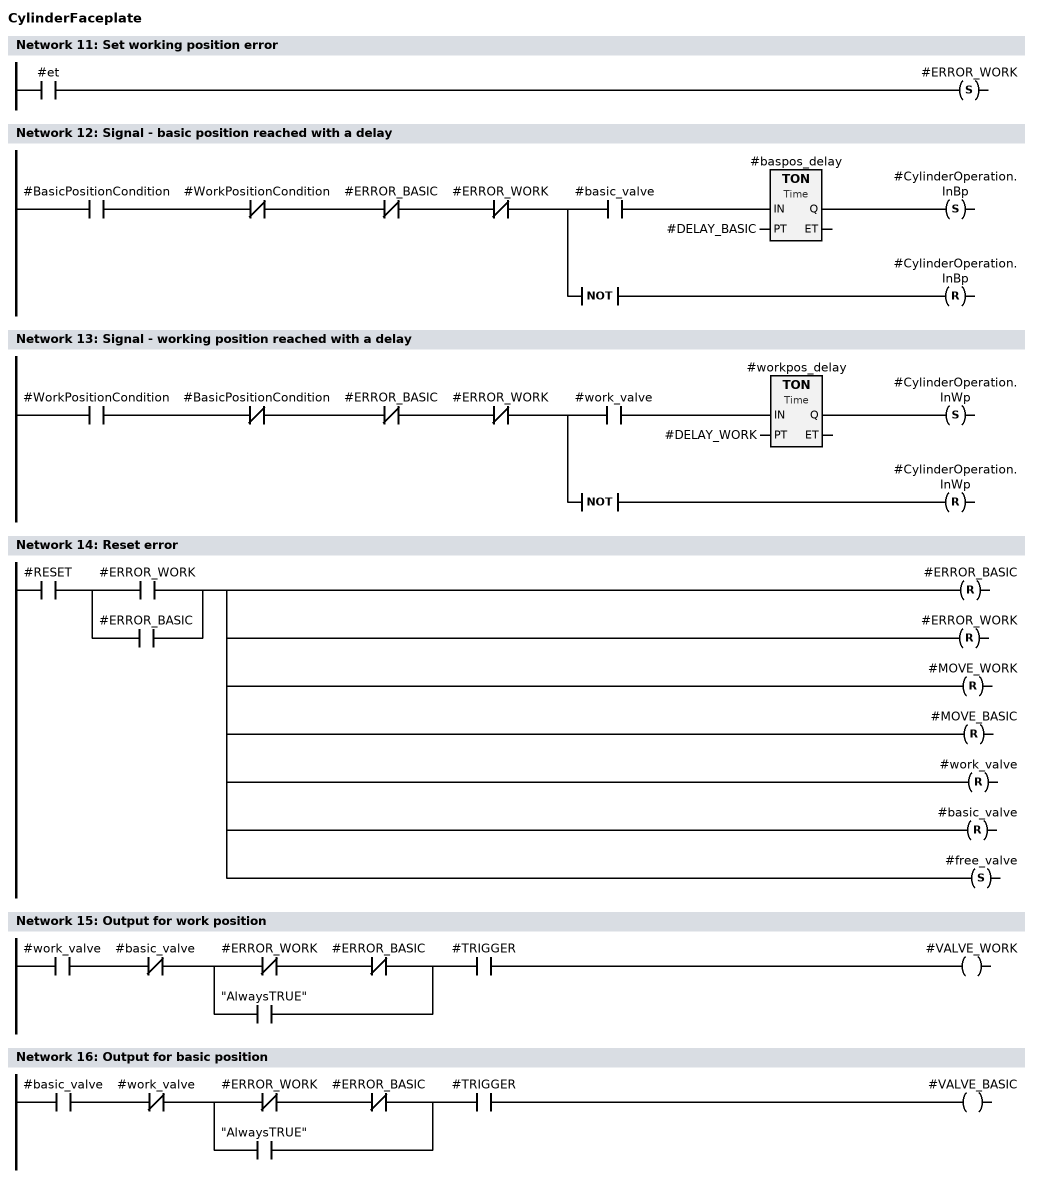
   RUNG wire#powerrail
      Contact( #et )
      S_Coil( #ERROR_WORK )
   END_RUNG
   // the same network as SCL:
   IF #et THEN #ERROR_WORK := TRUE; END_IF;
END_REGION

REGION Network 12: Signal - basic position reached with a delay
   RUNG wire#powerrail
      Contact( #BasicPositionCondition )
      I_Contact( #WorkPositionCondition )
      I_Contact( #ERROR_BASIC )
      I_Contact( #ERROR_WORK )
      wire#w1
      Contact( #basic_valve )
      { S7_Templates := "time_type := Time" } #baspos_delay.TON(pt := #DELAY_BASIC, et =>)
      S_Coil( #CylinderOperation.InBp )
   END_RUNG
   RUNG wire#w1
      Not()
      R_Coil( #CylinderOperation.InBp )
   END_RUNG
   // the same network as SCL:
   #_w1 := #BasicPositionCondition AND NOT #WorkPositionCondition AND NOT #ERROR_BASIC AND NOT #ERROR_WORK;
   #baspos_delay(IN := #_w1 AND #basic_valve, PT := #DELAY_BASIC);   // TON
   IF #baspos_delay.Q THEN #CylinderOperation.InBp := TRUE; END_IF;
   IF NOT #_w1 THEN #CylinderOperation.InBp := FALSE; END_IF;
END_REGION

REGION Network 13: Signal - working position reached with a delay
   RUNG wire#powerrail
      Contact( #WorkPositionCondition )
      I_Contact( #BasicPositionCondition )
      I_Contact( #ERROR_BASIC )
      I_Contact( #ERROR_WORK )
      wire#w1
      Contact( #work_valve )
      { S7_Templates := "time_type := Time" } #workpos_delay.TON(pt := #DELAY_WORK, et =>)
      S_Coil( #CylinderOperation.InWp )
   END_RUNG
   RUNG wire#w1
      Not()
      R_Coil( #CylinderOperation.InWp )
   END_RUNG
   // the same network as SCL:
   #_w1 := #WorkPositionCondition AND NOT #BasicPositionCondition AND NOT #ERROR_BASIC AND NOT #ERROR_WORK;
   #workpos_delay(IN := #_w1 AND #work_valve, PT := #DELAY_WORK);   // TON
   IF #workpos_delay.Q THEN #CylinderOperation.InWp := TRUE; END_IF;
   IF NOT #_w1 THEN #CylinderOperation.InWp := FALSE; END_IF;
END_REGION

REGION Network 14: Reset error
   RUNG wire#powerrail
      Contact( #RESET )
      wire#w1
      Contact( #ERROR_WORK )
      wire#w2
      R_Coil( #ERROR_BASIC )
   END_RUNG
   RUNG wire#w1
      Contact( #ERROR_BASIC )
   END_RUNG wire#w2
   RUNG wire#w2
      R_Coil( #ERROR_WORK )
   END_RUNG
   RUNG wire#w2
      R_Coil( #MOVE_WORK )
   END_RUNG
   RUNG wire#w2
      R_Coil( #MOVE_BASIC )
   END_RUNG
   RUNG wire#w2
      R_Coil( #work_valve )
   END_RUNG
   RUNG wire#w2
      R_Coil( #basic_valve )
   END_RUNG
   RUNG wire#w2
      S_Coil( #free_valve )
   END_RUNG
   // the same network as SCL:
   #_w1 := #RESET AND (#ERROR_WORK OR #ERROR_BASIC);
   IF #_w1 THEN
       #ERROR_BASIC := FALSE;
       #ERROR_WORK := FALSE;
       #MOVE_WORK := FALSE;
       #MOVE_BASIC := FALSE;
       #work_valve := FALSE;
       #basic_valve := FALSE;
       #free_valve := TRUE;
   END_IF;
END_REGION

REGION Network 15: Output for work position
   RUNG wire#powerrail
      Contact( #work_valve )
      I_Contact( #basic_valve )
      wire#w1
      I_Contact( #ERROR_WORK )
      I_Contact( #ERROR_BASIC )
      wire#w2
      Contact( #TRIGGER )
      Coil( #VALVE_WORK )
   END_RUNG
   RUNG wire#w1
      Contact( "AlwaysTRUE" )
   END_RUNG wire#w2
   // the same network as SCL:
   #VALVE_WORK := #work_valve AND NOT #basic_valve AND ((NOT #ERROR_WORK AND NOT #ERROR_BASIC) OR "AlwaysTRUE") AND #TRIGGER;
END_REGION

REGION Network 16: Output for basic position
   RUNG wire#powerrail
      Contact( #basic_valve )
      I_Contact( #work_valve )
      wire#w1
      I_Contact( #ERROR_WORK )
      I_Contact( #ERROR_BASIC )
      wire#w2
      Contact( #TRIGGER )
      Coil( #VALVE_BASIC )
   END_RUNG
   RUNG wire#w1
      Contact( "AlwaysTRUE" )
   END_RUNG wire#w2
   // the same network as SCL:
   #VALVE_BASIC := #basic_valve AND NOT #work_valve AND ((NOT #ERROR_WORK AND NOT #ERROR_BASIC) OR "AlwaysTRUE") AND #TRIGGER;
END_REGION

REGION Network 17 (SCL): Count status integer to HMI
   #comm := 0;
   IF #BasicPositionSensor THEN
       #comm := #comm + w#16#01;
   END_IF;

   IF #WorkPositionSensor THEN
       #comm := #comm + w#16#02;
   END_IF;

   IF #ERROR_BASIC THEN
       #comm := #comm + w#16#0040;
   END_IF;

   IF #ERROR_WORK THEN
       #comm := #comm + w#16#0080;
   END_IF;

   IF #VALVE_BASIC THEN
       #comm := #comm + w#16#0100;
   END_IF;
   IF #VALVE_WORK THEN
       #comm := #comm + w#16#0200;
   END_IF;

   IF NOT #iNoCollisionBasic THEN
       #comm := #comm + w#16#08;
   END_IF;

   IF NOT #iNoCollisionWork THEN
       #comm := #comm + w#16#10;
   END_IF;

   IF NOT #iNoCollisionFree THEN
       #comm := #comm + w#16#20;
   END_IF;

   #HMIStatus := #comm;
END_REGION
END_FUNCTION_BLOCK

FUNCTION_BLOCK "FittingCycle"   // FB35, LAD
{ S7_Optimized_Access := 'TRUE' }
VERSION : 0.1
// stored: AutoNumber true, IsIECCheckEnabled false, IsRetainMemResEnabled false, MemoryReserve 100, SetENOAutomatically false, UDAEnableTagReadback false
   VAR_INPUT
      parameters : "UDT_FittingParameters";
      basicPosition : Bool;
      MaxPosition : Real;
      endStopCylinderActive : Bool;
      shiftSupportToWork : Bool;
      rivetSensor : Bool;
      rivetStatusOtherCylinder : SInt;
   END_VAR
   VAR_IN_OUT
      HydraulicCylinder : "UDT_HydraulicCylinderData";
      dataFitting : "UDT_FittingStatus";
      dataDigiforce : "UDT_Digiforce";
      stopperForWedgeCylinder : "UDT_Cylinder";
      supportCylinder : "UDT_Cylinder";
      wedgeCylinder : "UDT_Cylinder";
      MeasuredData : "UDT_Results_Cupforming";
   END_VAR
   VAR
      cnt : Int;
      R_TRIG_Instance { S7_SetPoint := 'True'} : R_TRIG;
      H2Reached { S7_SetPoint := 'True'} : Bool;
      IEC_Timer_timeout { S7_SetPoint := 'True'} : TON_TIME;
      DigiforceStarted { S7_SetPoint := 'True'} : Bool;
      R_TRIG_Instance_1 { S7_SetPoint := 'True'} : R_TRIG;
      ton_WayWithTimeoutReached { S7_SetPoint := 'True'} : TON_TIME;
   END_VAR
   VAR_TEMP   // added for the SCL form of the ladder/FBD networks
      _w1 : Bool;
      _w2 : Bool;
   END_VAR
BEGIN

REGION Network 1: Check min max values
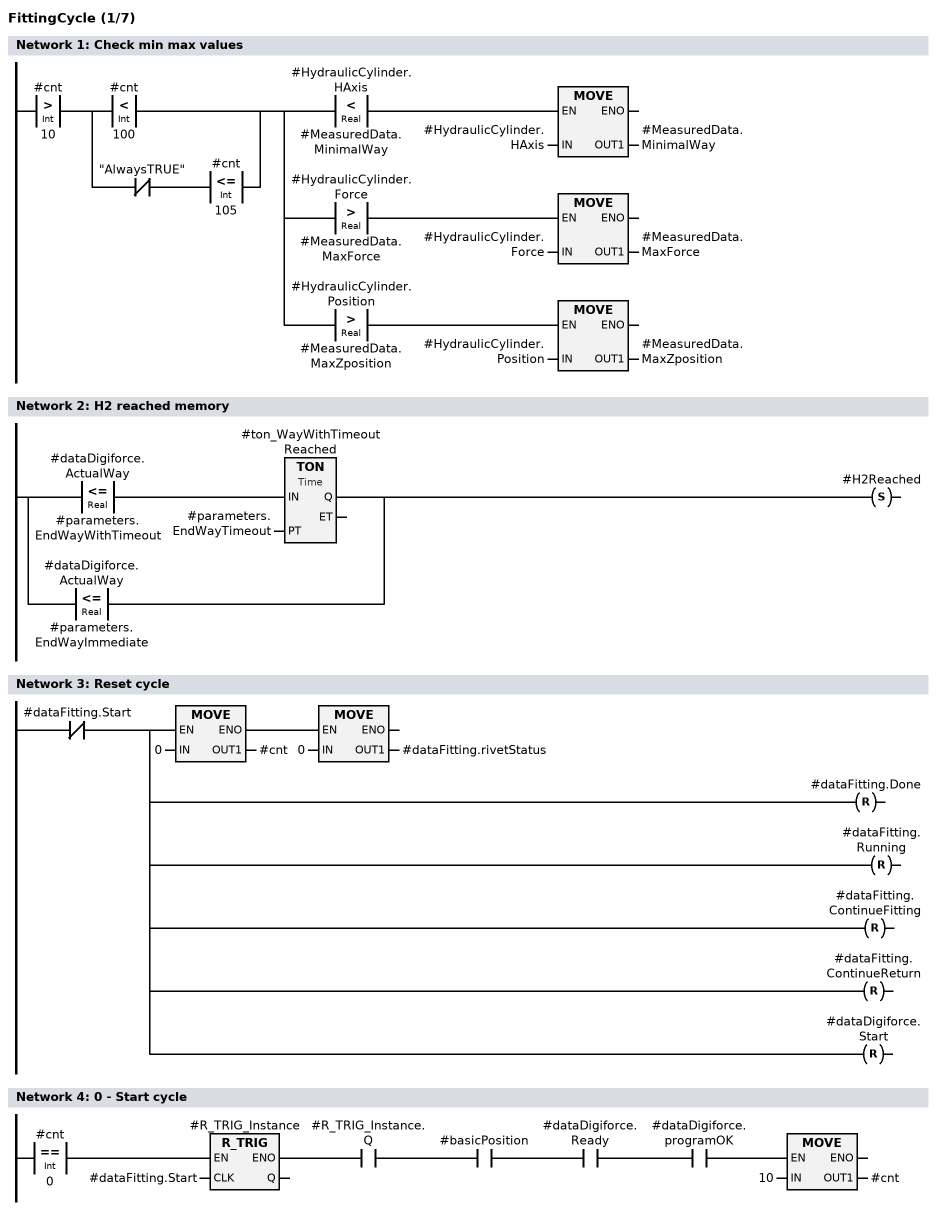
   RUNG wire#powerrail
      { S7_Templates := "SrcType := Int" } GT_Contact(in1 := #cnt, in2 := 10)
      wire#w1
      { S7_Templates := "SrcType := Int" } LT_Contact(in1 := #cnt, in2 := 100)
      wire#w2
      { S7_Templates := "SrcType := Real" } LT_Contact(in1 := #HydraulicCylinder.HAxis, in2 := #MeasuredData.MinimalWay)
      Move(in := #HydraulicCylinder.HAxis, out1 => #MeasuredData.MinimalWay)
   END_RUNG
   RUNG wire#w1
      I_Contact( "AlwaysTRUE" )
      { S7_Templates := "SrcType := Int" } LE_Contact(in1 := #cnt, in2 := 105)
   END_RUNG wire#w2
   RUNG wire#w2
      { S7_Templates := "SrcType := Real" } GT_Contact(in1 := #HydraulicCylinder.Force, in2 := #MeasuredData.MaxForce)
      Move(in := #HydraulicCylinder.Force, out1 => #MeasuredData.MaxForce)
   END_RUNG
   RUNG wire#w2
      { S7_Templates := "SrcType := Real" } GT_Contact(in1 := #HydraulicCylinder.Position, in2 := #MeasuredData.MaxZposition)
      Move(in := #HydraulicCylinder.Position, out1 => #MeasuredData.MaxZposition)
   END_RUNG
   // the same network as SCL:
   #_w1 := (#cnt > 10) AND ((#cnt < 100) OR (NOT "AlwaysTRUE" AND (#cnt <= 105)));
   IF #_w1 AND (#HydraulicCylinder.HAxis < #MeasuredData.MinimalWay) THEN
       #MeasuredData.MinimalWay := #HydraulicCylinder.HAxis;
   END_IF;
   IF #_w1 AND (#HydraulicCylinder.Force > #MeasuredData.MaxForce) THEN
       #MeasuredData.MaxForce := #HydraulicCylinder.Force;
   END_IF;
   IF #_w1 AND (#HydraulicCylinder.Position > #MeasuredData.MaxZposition) THEN
       #MeasuredData.MaxZposition := #HydraulicCylinder.Position;
   END_IF;
END_REGION

REGION Network 2: H2 reached memory
   RUNG wire#powerrail
      { S7_Templates := "SrcType := Real" } LE_Contact(in1 := #dataDigiforce.ActualWay, in2 := #parameters.EndWayWithTimeout)
      { S7_Templates := "time_type := Time" } #ton_WayWithTimeoutReached.TON(pt := #parameters.EndWayTimeout, et =>)
      wire#w1
      S_Coil( #H2Reached )
   END_RUNG
   RUNG wire#powerrail
      { S7_Templates := "SrcType := Real" } LE_Contact(in1 := #dataDigiforce.ActualWay, in2 := #parameters.EndWayImmediate)
   END_RUNG wire#w1
   // the same network as SCL:
   #ton_WayWithTimeoutReached(IN := #dataDigiforce.ActualWay <= #parameters.EndWayWithTimeout,   // TON
                           PT := #parameters.EndWayTimeout);
   IF #ton_WayWithTimeoutReached.Q OR (#dataDigiforce.ActualWay <= #parameters.EndWayImmediate) THEN
       #H2Reached := TRUE;
   END_IF;
END_REGION

REGION Network 3: Reset cycle
   RUNG wire#powerrail
      I_Contact( #dataFitting.Start )
      wire#w1
      Move(in := 0, out1 => #cnt)
      Move(in := 0, out1 => #dataFitting.rivetStatus)
   END_RUNG
   RUNG wire#w1
      R_Coil( #dataFitting.Done )
   END_RUNG
   RUNG wire#w1
      R_Coil( #dataFitting.Running )
   END_RUNG
   RUNG wire#w1
      R_Coil( #dataFitting.ContinueFitting )
   END_RUNG
   RUNG wire#w1
      R_Coil( #dataFitting.ContinueReturn )
   END_RUNG
   RUNG wire#w1
      R_Coil( #dataDigiforce.Start )
   END_RUNG
   // the same network as SCL:
   IF NOT #dataFitting.Start THEN
       #cnt := 0;
       #dataFitting.rivetStatus := 0;
       #dataFitting.Done := FALSE;
       #dataFitting.Running := FALSE;
       #dataFitting.ContinueFitting := FALSE;
       #dataFitting.ContinueReturn := FALSE;
       #dataDigiforce.Start := FALSE;
   END_IF;
END_REGION

REGION Network 4: 0 - Start cycle
   RUNG wire#powerrail
      { S7_Templates := "SrcType := Int" } EQ_Contact(in1 := #cnt, in2 := 0)
      #R_TRIG_Instance.R_TRIG(CLK := #dataFitting.Start, Q =>)
      Contact( #R_TRIG_Instance.Q )
      Contact( #basicPosition )
      Contact( #dataDigiforce.Ready )
      Contact( #dataDigiforce.programOK )
      Move(in := 10, out1 => #cnt)
   END_RUNG
   // the same network as SCL:
   #_w1 := #cnt = 0;
   #R_TRIG_Instance(EN := #_w1, CLK := #dataFitting.Start, ENO => #_w2);   // R_TRIG
   IF #_w2 AND #R_TRIG_Instance.Q AND #basicPosition AND #dataDigiforce.Ready AND #dataDigiforce.programOK THEN
       #cnt := 10;
   END_IF;
END_REGION

REGION Network 5: 10 - Start cycle
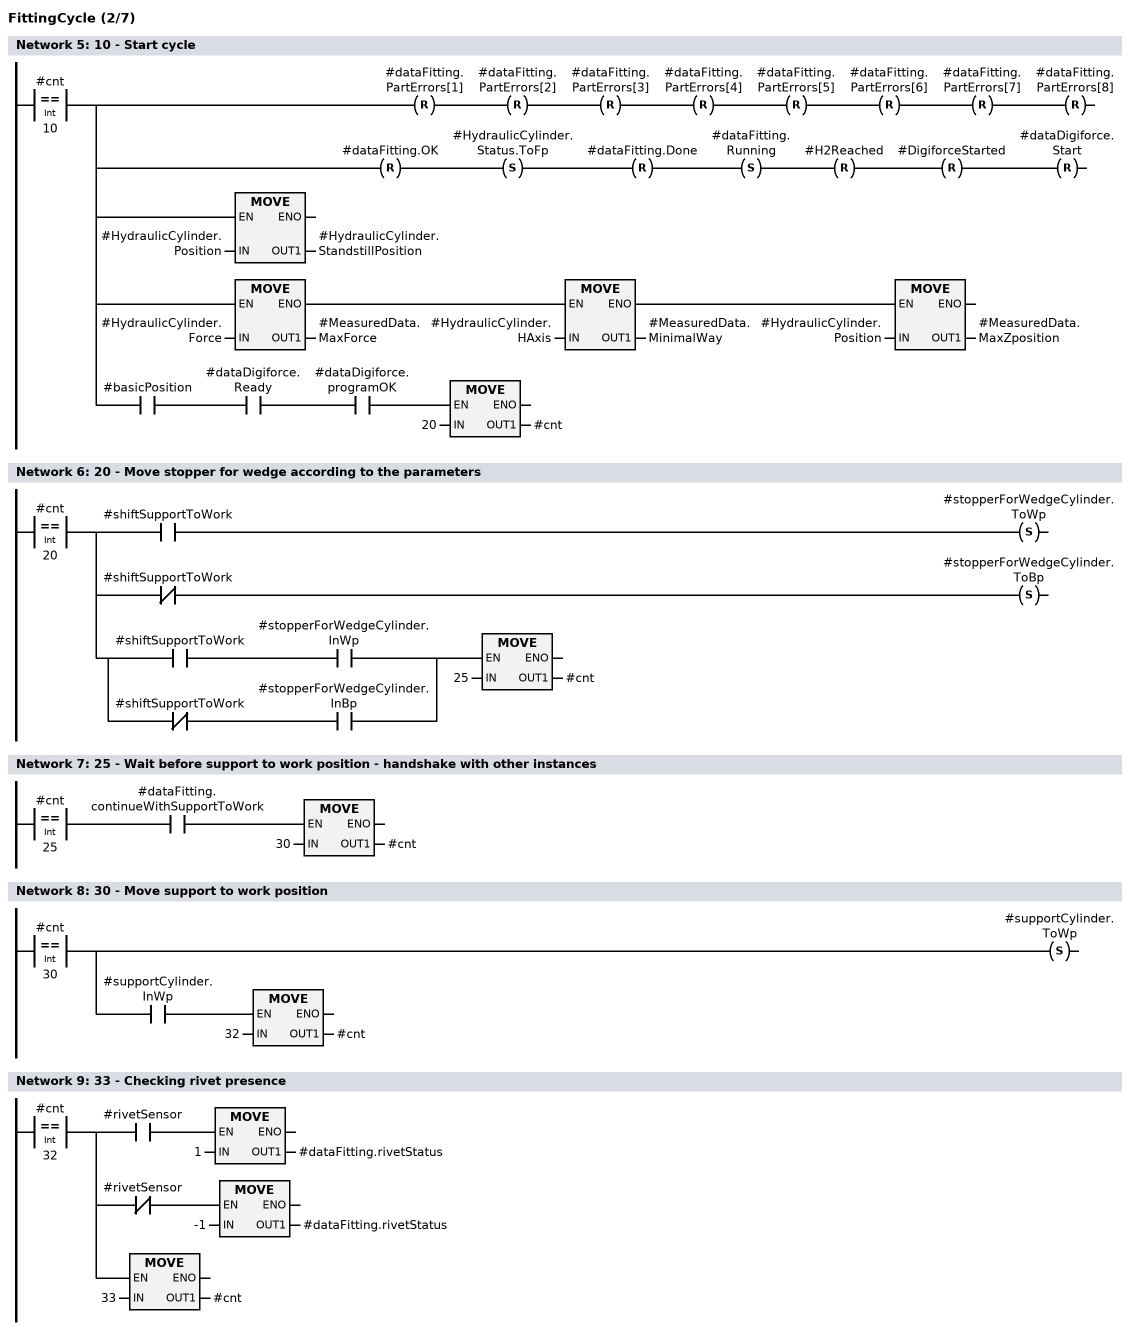
   RUNG wire#powerrail
      { S7_Templates := "SrcType := Int" } EQ_Contact(in1 := #cnt, in2 := 10)
      wire#w1
      R_Coil( #dataFitting.PartErrors[1] )
      R_Coil( #dataFitting.PartErrors[2] )
      R_Coil( #dataFitting.PartErrors[3] )
      R_Coil( #dataFitting.PartErrors[4] )
      R_Coil( #dataFitting.PartErrors[5] )
      R_Coil( #dataFitting.PartErrors[6] )
      R_Coil( #dataFitting.PartErrors[7] )
      R_Coil( #dataFitting.PartErrors[8] )
   END_RUNG
   RUNG wire#w1
      R_Coil( #dataFitting.OK )
      S_Coil( #HydraulicCylinder.Status.ToFp )
      R_Coil( #dataFitting.Done )
      S_Coil( #dataFitting.Running )
      R_Coil( #H2Reached )
      R_Coil( #DigiforceStarted )
      R_Coil( #dataDigiforce.Start )
   END_RUNG
   RUNG wire#w1
      Move(in := #HydraulicCylinder.Position, out1 => #HydraulicCylinder.StandstillPosition)
   END_RUNG
   RUNG wire#w1
      Move(in := #HydraulicCylinder.Force, out1 => #MeasuredData.MaxForce)
      Move(in := #HydraulicCylinder.HAxis, out1 => #MeasuredData.MinimalWay)
      Move(in := #HydraulicCylinder.Position, out1 => #MeasuredData.MaxZposition)
   END_RUNG
   RUNG wire#w1
      Contact( #basicPosition )
      Contact( #dataDigiforce.Ready )
      Contact( #dataDigiforce.programOK )
      Move(in := 20, out1 => #cnt)
   END_RUNG
   // the same network as SCL:
   #_w1 := #cnt = 10;
   IF #_w1 THEN
       #dataFitting.PartErrors[1] := FALSE;
       #dataFitting.PartErrors[2] := FALSE;
       #dataFitting.PartErrors[3] := FALSE;
       #dataFitting.PartErrors[4] := FALSE;
       #dataFitting.PartErrors[5] := FALSE;
       #dataFitting.PartErrors[6] := FALSE;
       #dataFitting.PartErrors[7] := FALSE;
       #dataFitting.PartErrors[8] := FALSE;
       #dataFitting.OK := FALSE;
       #HydraulicCylinder.Status.ToFp := TRUE;
       #dataFitting.Done := FALSE;
       #dataFitting.Running := TRUE;
       #H2Reached := FALSE;
       #DigiforceStarted := FALSE;
       #dataDigiforce.Start := FALSE;
       #HydraulicCylinder.StandstillPosition := #HydraulicCylinder.Position;
       #MeasuredData.MaxForce := #HydraulicCylinder.Force;
       #MeasuredData.MinimalWay := #HydraulicCylinder.HAxis;
       #MeasuredData.MaxZposition := #HydraulicCylinder.Position;
   END_IF;
   IF #_w1 AND #basicPosition AND #dataDigiforce.Ready AND #dataDigiforce.programOK THEN #cnt := 20; END_IF;
END_REGION

REGION Network 6: 20 - Move stopper for wedge according to the parameters
   RUNG wire#powerrail
      { S7_Templates := "SrcType := Int" } EQ_Contact(in1 := #cnt, in2 := 20)
      wire#w1
      Contact( #shiftSupportToWork )
      S_Coil( #stopperForWedgeCylinder.ToWp )
   END_RUNG
   RUNG wire#w1
      I_Contact( #shiftSupportToWork )
      S_Coil( #stopperForWedgeCylinder.ToBp )
   END_RUNG
   RUNG wire#w1
      Contact( #shiftSupportToWork )
      Contact( #stopperForWedgeCylinder.InWp )
      wire#w2
      Move(in := 25, out1 => #cnt)
   END_RUNG
   RUNG wire#w1
      I_Contact( #shiftSupportToWork )
      Contact( #stopperForWedgeCylinder.InBp )
   END_RUNG wire#w2
   // the same network as SCL:
   #_w1 := #cnt = 20;
   IF #_w1 AND #shiftSupportToWork THEN #stopperForWedgeCylinder.ToWp := TRUE; END_IF;
   IF #_w1 AND NOT #shiftSupportToWork THEN #stopperForWedgeCylinder.ToBp := TRUE; END_IF;
   IF #_w1 AND ((#shiftSupportToWork AND #stopperForWedgeCylinder.InWp) OR (NOT #shiftSupportToWork AND #stopperForWedgeCylinder.InBp)) THEN
       #cnt := 25;
   END_IF;
END_REGION

REGION Network 7: 25 - Wait before support to work position - handshake with other instances
   RUNG wire#powerrail
      { S7_Templates := "SrcType := Int" } EQ_Contact(in1 := #cnt, in2 := 25)
      Contact( #dataFitting.continueWithSupportToWork )
      Move(in := 30, out1 => #cnt)
   END_RUNG
   // the same network as SCL:
   IF (#cnt = 25) AND #dataFitting.continueWithSupportToWork THEN #cnt := 30; END_IF;
END_REGION

REGION Network 8: 30 - Move support to work position
   RUNG wire#powerrail
      { S7_Templates := "SrcType := Int" } EQ_Contact(in1 := #cnt, in2 := 30)
      wire#w1
      S_Coil( #supportCylinder.ToWp )
   END_RUNG
   RUNG wire#w1
      Contact( #supportCylinder.InWp )
      Move(in := 32, out1 => #cnt)
   END_RUNG
   // the same network as SCL:
   #_w1 := #cnt = 30;
   IF #_w1 THEN #supportCylinder.ToWp := TRUE; END_IF;
   IF #_w1 AND #supportCylinder.InWp THEN #cnt := 32; END_IF;
END_REGION

REGION Network 9: 33 - Checking rivet presence
   RUNG wire#powerrail
      { S7_Templates := "SrcType := Int" } EQ_Contact(in1 := #cnt, in2 := 32)
      wire#w1
      Contact( #rivetSensor )
      Move(in := 1, out1 => #dataFitting.rivetStatus)
   END_RUNG
   RUNG wire#w1
      I_Contact( #rivetSensor )
      Move(in := -1, out1 => #dataFitting.rivetStatus)
   END_RUNG
   RUNG wire#w1
      Move(in := 33, out1 => #cnt)
   END_RUNG
   // the same network as SCL:
   #_w1 := #cnt = 32;
   IF #_w1 AND #rivetSensor THEN #dataFitting.rivetStatus := 1; END_IF;
   IF #_w1 AND NOT #rivetSensor THEN #dataFitting.rivetStatus := -1; END_IF;
   IF #_w1 THEN #cnt := 33; END_IF;
END_REGION

REGION Network 10: 34 - Rivet presence result / handshake
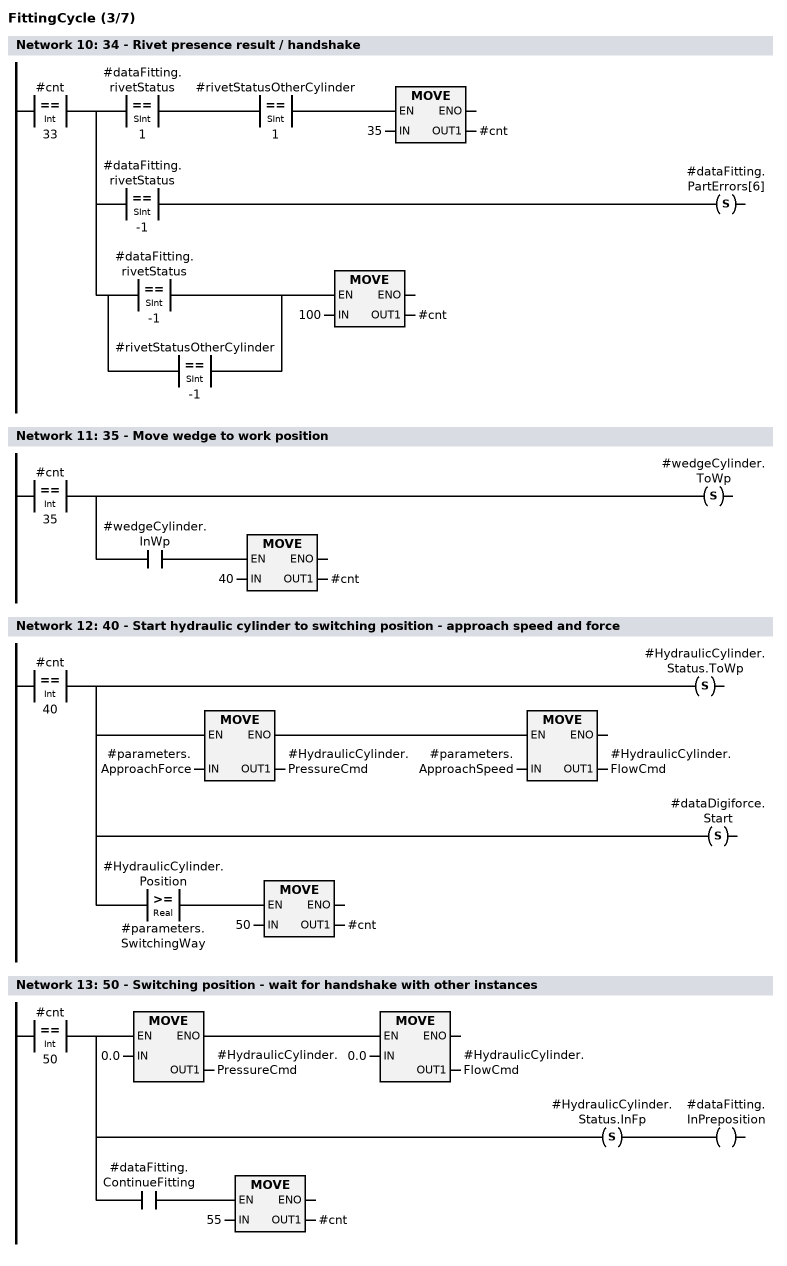
   RUNG wire#powerrail
      { S7_Templates := "SrcType := Int" } EQ_Contact(in1 := #cnt, in2 := 33)
      wire#w1
      { S7_Templates := "SrcType := SInt" } EQ_Contact(in1 := #dataFitting.rivetStatus, in2 := 1)
      { S7_Templates := "SrcType := SInt" } EQ_Contact(in1 := #rivetStatusOtherCylinder, in2 := 1)
      Move(in := 35, out1 => #cnt)
   END_RUNG
   RUNG wire#w1
      { S7_Templates := "SrcType := SInt" } EQ_Contact(in1 := #dataFitting.rivetStatus, in2 := -1)
      S_Coil( #dataFitting.PartErrors[6] )
   END_RUNG
   RUNG wire#w1
      { S7_Templates := "SrcType := SInt" } EQ_Contact(in1 := #dataFitting.rivetStatus, in2 := -1)
      wire#w2
      Move(in := 100, out1 => #cnt)
   END_RUNG
   RUNG wire#w1
      { S7_Templates := "SrcType := SInt" } EQ_Contact(in1 := #rivetStatusOtherCylinder, in2 := -1)
   END_RUNG wire#w2
   // the same network as SCL:
   #_w1 := #cnt = 33;
   IF #_w1 AND (#dataFitting.rivetStatus = 1) AND (#rivetStatusOtherCylinder = 1) THEN #cnt := 35; END_IF;
   IF #_w1 AND (#dataFitting.rivetStatus = (-1)) THEN #dataFitting.PartErrors[6] := TRUE; END_IF;
   IF #_w1 AND ((#dataFitting.rivetStatus = (-1)) OR (#rivetStatusOtherCylinder = (-1))) THEN
       #cnt := 100;
   END_IF;
END_REGION

REGION Network 11: 35 - Move wedge to work position
   RUNG wire#powerrail
      { S7_Templates := "SrcType := Int" } EQ_Contact(in1 := #cnt, in2 := 35)
      wire#w1
      S_Coil( #wedgeCylinder.ToWp )
   END_RUNG
   RUNG wire#w1
      Contact( #wedgeCylinder.InWp )
      Move(in := 40, out1 => #cnt)
   END_RUNG
   // the same network as SCL:
   #_w1 := #cnt = 35;
   IF #_w1 THEN #wedgeCylinder.ToWp := TRUE; END_IF;
   IF #_w1 AND #wedgeCylinder.InWp THEN #cnt := 40; END_IF;
END_REGION

REGION Network 12: 40 - Start hydraulic cylinder to switching position - approach speed and force
   RUNG wire#powerrail
      { S7_Templates := "SrcType := Int" } EQ_Contact(in1 := #cnt, in2 := 40)
      wire#w1
      S_Coil( #HydraulicCylinder.Status.ToWp )
   END_RUNG
   RUNG wire#w1
      Move(in := #parameters.ApproachForce, out1 => #HydraulicCylinder.PressureCmd)
      Move(in := #parameters.ApproachSpeed, out1 => #HydraulicCylinder.FlowCmd)
   END_RUNG
   RUNG wire#w1
      S_Coil( #dataDigiforce.Start )
   END_RUNG
   RUNG wire#w1
      { S7_Templates := "SrcType := Real" } GE_Contact(in1 := #HydraulicCylinder.Position, in2 := #parameters.SwitchingWay)
      Move(in := 50, out1 => #cnt)
   END_RUNG
   // the same network as SCL:
   #_w1 := #cnt = 40;
   IF #_w1 THEN
       #HydraulicCylinder.Status.ToWp := TRUE;
       #HydraulicCylinder.PressureCmd := #parameters.ApproachForce;
       #HydraulicCylinder.FlowCmd := #parameters.ApproachSpeed;
       #dataDigiforce.Start := TRUE;
   END_IF;
   IF #_w1 AND (#HydraulicCylinder.Position >= #parameters.SwitchingWay) THEN #cnt := 50; END_IF;
END_REGION

REGION Network 13: 50 - Switching position - wait for handshake with other instances
   RUNG wire#powerrail
      { S7_Templates := "SrcType := Int" } EQ_Contact(in1 := #cnt, in2 := 50)
      wire#w1
      Move(in := 0.0, out1 => #HydraulicCylinder.PressureCmd)
      Move(in := 0.0, out1 => #HydraulicCylinder.FlowCmd)
   END_RUNG
   RUNG wire#w1
      S_Coil( #HydraulicCylinder.Status.InFp )
      Coil( #dataFitting.InPreposition )
   END_RUNG
   RUNG wire#w1
      Contact( #dataFitting.ContinueFitting )
      Move(in := 55, out1 => #cnt)
   END_RUNG
   // the same network as SCL:
   #_w1 := #cnt = 50;
   IF #_w1 THEN
       #HydraulicCylinder.PressureCmd := 0.0;
       #HydraulicCylinder.FlowCmd := 0.0;
       #HydraulicCylinder.Status.InFp := TRUE;
   END_IF;
   #dataFitting.InPreposition := #_w1;
   IF #_w1 AND #dataFitting.ContinueFitting THEN #cnt := 55; END_IF;
END_REGION

REGION Network 14: 55 - Move sidemember to work position
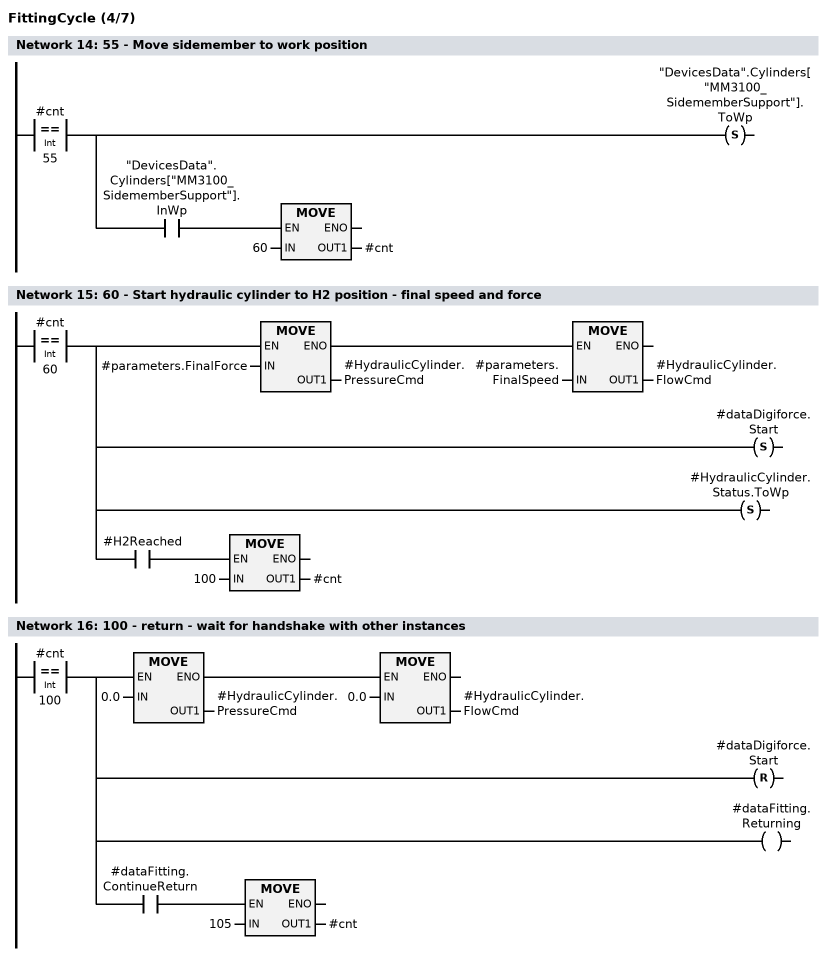
   RUNG wire#powerrail
      { S7_Templates := "SrcType := Int" } EQ_Contact(in1 := #cnt, in2 := 55)
      wire#w1
      S_Coil( "DevicesData".Cylinders["MM3100_SidememberSupport"].ToWp )
   END_RUNG
   RUNG wire#w1
      Contact( "DevicesData".Cylinders["MM3100_SidememberSupport"].InWp )
      Move(in := 60, out1 => #cnt)
   END_RUNG
   // the same network as SCL:
   #_w1 := #cnt = 55;
   IF #_w1 THEN "DevicesData".Cylinders["MM3100_SidememberSupport"].ToWp := TRUE; END_IF;
   IF #_w1 AND "DevicesData".Cylinders["MM3100_SidememberSupport"].InWp THEN #cnt := 60; END_IF;
END_REGION

REGION Network 15: 60 - Start hydraulic cylinder to H2 position - final speed and force
   RUNG wire#powerrail
      { S7_Templates := "SrcType := Int" } EQ_Contact(in1 := #cnt, in2 := 60)
      wire#w1
      Move(in := #parameters.FinalForce, out1 => #HydraulicCylinder.PressureCmd)
      Move(in := #parameters.FinalSpeed, out1 => #HydraulicCylinder.FlowCmd)
   END_RUNG
   RUNG wire#w1
      S_Coil( #dataDigiforce.Start )
   END_RUNG
   RUNG wire#w1
      S_Coil( #HydraulicCylinder.Status.ToWp )
   END_RUNG
   RUNG wire#w1
      Contact( #H2Reached )
      Move(in := 100, out1 => #cnt)
   END_RUNG
   // the same network as SCL:
   #_w1 := #cnt = 60;
   IF #_w1 THEN
       #HydraulicCylinder.PressureCmd := #parameters.FinalForce;
       #HydraulicCylinder.FlowCmd := #parameters.FinalSpeed;
       #dataDigiforce.Start := TRUE;
       #HydraulicCylinder.Status.ToWp := TRUE;
   END_IF;
   IF #_w1 AND #H2Reached THEN #cnt := 100; END_IF;
END_REGION

